LIN {X 0,Y 161.237,Z 153.823,A -85,B 0,C 180,E1 -25905.444,E2 -25905.444} C_VEL
LIN {X 0,Y 158.959,Z 150.146,A -85,B 0,C 180,E1 -25908.846,E2 -25908.846} C_VEL
LIN {X 0,Y 156.887,Z 147.156,A -85,B 0,C 180,E1 -25912.883,E2 -25912.883} C_VEL
LIN {X 0,Y 156.329,Z 145.593,A -85,B 0,C 180,E1 -25914.517,E2 -25914.517} C_VEL
LIN {X 0,Y 154.928,Z 144.258,A -85,B 0,C 180,E1 -25919.999,E2 -25919.999} C_VEL
LIN {X 0,Y 154.751,Z 144.476,A -85,B 0,C 180,E1 -25925.211,E2 -25925.211} C_VEL
LIN {X 0,Y 156.305,Z 145.838,A -85,B 0,C 180,E1 -25931.923,E2 -25931.923} C_VEL
LIN {X 0,Y 158.287,Z 149.53,A -85,B 0,C 180,E1 -25936.483,E2 -25936.483} C_VEL
LIN {X 0,Y 159.389,Z 150.896,A -85,B 0,C 180,E1 -25938.299,E2 -25938.299} C_VEL
LIN {X 0,Y 161.903,Z 155.182,A -85,B 0,C 180,E1 -25941.881,E2 -25941.881} C_VEL
LIN {X 0,Y 164.505,Z 160.547,A -85,B 0,C 180,E1 -25945.01,E2 -25945.01} C_VEL
LIN {X 0,Y 167.627,Z 167.381,A -85,B 0,C 180,E1 -25948.21,E2 -25948.21} C_VEL
LIN {X 0,Y 171.486,Z 176.831,A -85,B 0,C 180,E1 -25951.653,E2 -25951.653} C_VEL
LIN {X 0,Y 174.833,Z 186.302,A -85,B 0,C 180,E1 -25954.344,E2 -25954.344} C_VEL
LIN {X 0,Y 172.854,Z 207.577,A -85,B 0,C 180,E1 -25955.092,E2 -25955.092} C_VEL
LIN {X 0,Y 170.404,Z 220.728,A -85,B 0,C 180,E1 -25955.779,E2 -25955.779} C_VEL
LIN {X 0,Y 167.271,Z 232.382,A -85,B 0,C 180,E1 -25956.695,E2 -25956.695} C_VEL
LIN {X 0,Y 162.827,Z 244.666,A -85,B 0,C 180,E1 -25958.027,E2 -25958.027} C_VEL
LIN {X 0,Y 157.562,Z 256.097,A -85,B 0,C 180,E1 -25959.696,E2 -25959.696} C_VEL
LIN {X 0,Y 151.989,Z 266.408,A -85,B 0,C 180,E1 -25961.786,E2 -25961.786} C_VEL
LIN {X 0,Y 146.595,Z 274.853,A -85,B 0,C 180,E1 -25964.017,E2 -25964.017} C_VEL
LIN {X 0,Y 139.883,Z 284.024,A -85,B 0,C 180,E1 -25967.291,E2 -25967.291} C_VEL
LIN {X 0,Y 133.694,Z 291.425,A -85,B 0,C 180,E1 -25970.889,E2 -25970.889} C_VEL
LIN {X 0,Y 128.246,Z 297.387,A -85,B 0,C 180,E1 -25974.87,E2 -25974.87} C_VEL
LIN {X 0,Y 123.535,Z 302.12,A -85,B 0,C 180,E1 -25979.201,E2 -25979.201} C_VEL
LIN {X 0,Y 119.473,Z 305.757,A -85,B 0,C 180,E1 -25983.819,E2 -25983.819} C_VEL
LIN {X 0,Y 116.246,Z 308.403,A -85,B 0,C 180,E1 -25988.73,E2 -25988.73} C_VEL
LIN {X 0,Y 114.629,Z 309.67,A -85,B 0,C 180,E1 -25992.147,E2 -25992.147} C_VEL
LIN {X 0,Y 113.509,Z 310.529,A -85,B 0,C 180,E1 -25995.66,E2 -25995.66} C_VEL
LIN {X 0,Y 112.333,Z 311.033,A -85,B 0,C 180,E1 -26002.811,E2 -26002.811} C_VEL
LIN {X 0,Y 112.458,Z 310.179,A -85,B 0,C 180,E1 -26009.194,E2 -26009.194} C_VEL
LIN {X 0,Y 112.346,Z 308.795,A -85,B 0,C 180,E1 -26013.586,E2 -26013.586} C_VEL
LIN {X 0,Y 112.488,Z 306.212,A -85,B 0,C 180,E1 -26018.985,E2 -26018.985} C_VEL
LIN {X 0,Y 113.368,Z 302.594,A -85,B 0,C 180,E1 -26024.356,E2 -26024.356} C_VEL
LIN {X 0,Y 115.16,Z 297.853,A -85,B 0,C 180,E1 -26029.611,E2 -26029.611} C_VEL
LIN {X 0,Y 117.825,Z 291.844,A -85,B 0,C 180,E1 -26034.678,E2 -26034.678} C_VEL
LIN {X 0,Y 120.577,Z 286.067,A -85,B 0,C 180,E1 -26038.505,E2 -26038.505} C_VEL
LIN {X 0,Y 124.02,Z 278.346,A -85,B 0,C 180,E1 -26042.57,E2 -26042.57} C_VEL
LIN {X 0,Y 126.266,Z 273.338,A -85,B 0,C 180,E1 -26044.711,E2 -26044.711} C_VEL
LIN {X 0,Y 127.579,Z 269.067,A -85,B 0,C 180,E1 -26046.467,E2 -26046.467} C_VEL
LIN {X 0,Y 128.278,Z 261.803,A -85,B 0,C 180,E1 -26049.488,E2 -26049.488} C_VEL
LIN {X 0,Y 129.024,Z 254.081,A -85,B 0,C 180,E1 -26052.242,E2 -26052.242} C_VEL
LIN {X 0,Y 130.33,Z 249.097,A -85,B 0,C 180,E1 -26053.522,E2 -26053.522} C_VEL
LIN {X 0,Y 134.094,Z 237.597,A -85,B 0,C 180,E1 -26055.568,E2 -26055.568} C_VEL
LIN {X 0,Y 137.193,Z 225.349,A -85,B 0,C 180,E1 -26057.153,E2 -26057.153} C_VEL
LIN {X 0,Y 139.495,Z 212.87,A -85,B 0,C 180,E1 -26058.268,E2 -26058.268} C_VEL
LIN {X 0,Y 140.933,Z 199.169,A -85,B 0,C 180,E1 -26059.042,E2 -26059.042} C_VEL
LIN {X 0,Y 143.055,Z 169.052,A -85,B 0,C 180,E1 -26060.308,E2 -26060.308} C_VEL
LIN {X 0,Y 142.696,Z 161.497,A -85,B 0,C 180,E1 -26061.009,E2 -26061.009} C_VEL
LIN {X 0,Y 139.659,Z 152.428,A -85,B 0,C 180,E1 -26063.079,E2 -26063.079} C_VEL
LIN {X 0,Y 135.374,Z 142.008,A -85,B 0,C 180,E1 -26066.124,E2 -26066.124} C_VEL
LIN {X 0,Y 132.711,Z 136.591,A -85,B 0,C 180,E1 -26068.136,E2 -26068.136} C_VEL
LIN {X 0,Y 127.721,Z 129.053,A -85,B 0,C 180,E1 -26072.186,E2 -26072.186} C_VEL
LIN {X 0,Y 124.838,Z 124.988,A -85,B 0,C 180,E1 -26074.886,E2 -26074.886} C_VEL
LIN {X 0,Y 122.223,Z 121.297,A -85,B 0,C 180,E1 -26077.677,E2 -26077.677} C_VEL
LIN {X 0,Y 119.05,Z 117.651,A -85,B 0,C 180,E1 -26081.556,E2 -26081.556} C_VEL
LIN {X 0,Y 118.034,Z 115.687,A -85,B 0,C 180,E1 -26083.127,E2 -26083.127} C_VEL
LIN {X 0,Y 115.584,Z 113.816,A -85,B 0,C 180,E1 -26087.028,E2 -26087.028} C_VEL
LIN {X 0,Y 114.038,Z 110.593,A -85,B 0,C 180,E1 -26090.692,E2 -26090.692} C_VEL
LIN {X 0,Y 113.905,Z 110.069,A -85,B 0,C 180,E1 -26091.129,E2 -26091.129} C_VEL
LIN {X 0,Y 111.558,Z 108.57,A -85,B 0,C 180,E1 -26100.001,E2 -26100.001} C_VEL
LIN {X 0,Y 112.791,Z 109.816,A -85,B 0,C 180,E1 -26113.637,E2 -26113.637} C_VEL
LIN {X 0,Y 113.656,Z 110.24,A -85,B 0,C 180,E1 -26116.042,E2 -26116.042} C_VEL
LIN {X 0,Y 114.742,Z 112.902,A -85,B 0,C 180,E1 -26118.99,E2 -26118.99} C_VEL
LIN {X 0,Y 117.084,Z 115.281,A -85,B 0,C 180,E1 -26123.218,E2 -26123.218} C_VEL
LIN {X 0,Y 118.127,Z 115.966,A -85,B 0,C 180,E1 -26124.73,E2 -26124.73} C_VEL
LIN {X 0,Y 120.133,Z 119.302,A -85,B 0,C 180,E1 -26127.611,E2 -26127.611} C_VEL
LIN {X 0,Y 122.237,Z 121.386,A -85,B 0,C 180,E1 -26130.044,E2 -26130.044} C_VEL
LIN {X 0,Y 124.625,Z 124.868,A -85,B 0,C 180,E1 -26132.619,E2 -26132.619} C_VEL
LIN {X 0,Y 125.763,Z 126.328,A -85,B 0,C 180,E1 -26133.72,E2 -26133.72} C_VEL
LIN {X 0,Y 129.511,Z 131.842,A -85,B 0,C 180,E1 -26137.059,E2 -26137.059} C_VEL
LIN {X 0,Y 133.457,Z 137.926,A -85,B 0,C 180,E1 -26140.126,E2 -26140.126} C_VEL
LIN {X 0,Y 138.292,Z 146.234,A -85,B 0,C 180,E1 -26143.461,E2 -26143.461} C_VEL
LIN {X 0,Y 142.745,Z 155.217,A -85,B 0,C 180,E1 -26146.252,E2 -26146.252} C_VEL
LIN {X 0,Y 143.805,Z 157.638,A -85,B 0,C 180,E1 -26146.891,E2 -26146.891} C_VEL
LIN {X 0,Y 140.743,Z 198.449,A -85,B 0,C 180,E1 -26148.657,E2 -26148.657} C_VEL
LIN {X 0,Y 138.718,Z 212.325,A -85,B 0,C 180,E1 -26149.763,E2 -26149.763} C_VEL
LIN {X 0,Y 136.225,Z 224.495,A -85,B 0,C 180,E1 -26151.279,E2 -26151.279} C_VEL
LIN {X 0,Y 132.73,Z 237.021,A -85,B 0,C 180,E1 -26153.44,E2 -26153.44} C_VEL
LIN {X 0,Y 128.857,Z 248.183,A -85,B 0,C 180,E1 -26156.011,E2 -26156.011} C_VEL
LIN {X 0,Y 124.728,Z 258.248,A -85,B 0,C 180,E1 -26159.06,E2 -26159.06} C_VEL
LIN {X 0,Y 120.096,Z 268.136,A -85,B 0,C 180,E1 -26163.031,E2 -26163.031} C_VEL
LIN {X 0,Y 115.725,Z 276.841,A -85,B 0,C 180,E1 -26167.694,E2 -26167.694} C_VEL
LIN {X 0,Y 112.073,Z 283.795,A -85,B 0,C 180,E1 -26172.671,E2 -26172.671} C_VEL
LIN {X 0,Y 108.756,Z 290.167,A -85,B 0,C 180,E1 -26178.823,E2 -26178.823} C_VEL
LIN {X 0,Y 106.899,Z 294.363,A -85,B 0,C 180,E1 -26184.342,E2 -26184.342} C_VEL
LIN {X 0,Y 105.799,Z 297.516,A -85,B 0,C 180,E1 -26190.001,E2 -26190.001} C_VEL
LIN {X 0,Y 105.513,Z 299.091,A -85,B 0,C 180,E1 -26193.82,E2 -26193.82} C_VEL
LIN {X 0,Y 105.334,Z 300.263,A -85,B 0,C 180,E1 -26197.67,E2 -26197.67} C_VEL
LIN {X 0,Y 106.07,Z 301.363,A -85,B 0,C 180,E1 -26205.37,E2 -26205.37} C_VEL
LIN {X 0,Y 107.02,Z 301.338,A -85,B 0,C 180,E1 -26209.17,E2 -26209.17} C_VEL
LIN {X 0,Y 108.419,Z 300.902,A -85,B 0,C 180,E1 -26212.889,E2 -26212.889} C_VEL
LIN {X 0,Y 110.561,Z 299.844,A -85,B 0,C 180,E1 -26217.133,E2 -26217.133} C_VEL
LIN {X 0,Y 114.79,Z 297.11,A -85,B 0,C 180,E1 -26223.439,E2 -26223.439} C_VEL
LIN {X 0,Y 119.167,Z 293.727,A -85,B 0,C 180,E1 -26228.263,E2 -26228.263} C_VEL
LIN {X 0,Y 124.307,Z 289.239,A -85,B 0,C 180,E1 -26232.724,E2 -26232.724} C_VEL
LIN {X 0,Y 131.157,Z 282.378,A -85,B 0,C 180,E1 -26237.46,E2 -26237.46} C_VEL
LIN {X 0,Y 137.67,Z 274.904,A -85,B 0,C 180,E1 -26241.125,E2 -26241.125} C_VEL
LIN {X 0,Y 143.894,Z 266.42,A -85,B 0,C 180,E1 -26244.283,E2 -26244.283} C_VEL
LIN {X 0,Y 149.993,Z 256.814,A -85,B 0,C 180,E1 -26246.883,E2 -26246.883} C_VEL
LIN {X 0,Y 155.772,Z 246.135,A -85,B 0,C 180,E1 -26249.009,E2 -26249.009} C_VEL
LIN {X 0,Y 160.389,Z 235.789,A -85,B 0,C 180,E1 -26250.564,E2 -26250.564} C_VEL
LIN {X 0,Y 164.457,Z 224.001,A -85,B 0,C 180,E1 -26251.96,E2 -26251.96} C_VEL
LIN {X 0,Y 167.84,Z 211.19,A -85,B 0,C 180,E1 -26252.975,E2 -26252.975} C_VEL
LIN {X 0,Y 170.071,Z 198.637,A -85,B 0,C 180,E1 -26253.644,E2 -26253.644} C_VEL
LIN {X 0,Y 171.608,Z 182.647,A -85,B 0,C 180,E1 -26254.204,E2 -26254.204} C_VEL
LIN {X 0,Y 167.577,Z 174.242,A -85,B 0,C 180,E1 -26257.58,E2 -26257.58} C_VEL
LIN {X 0,Y 163.832,Z 167.391,A -85,B 0,C 180,E1 -26261.211,E2 -26261.211} C_VEL
LIN {X 0,Y 161.108,Z 162.795,A -85,B 0,C 180,E1 -26264.34,E2 -26264.34} C_VEL
LIN {X 0,Y 159.533,Z 160.138,A -85,B 0,C 180,E1 -26266.465,E2 -26266.465} C_VEL
LIN {X 0,Y 157.704,Z 156.967,A -85,B 0,C 180,E1 -26269.407,E2 -26269.407} C_VEL
LIN {X 0,Y 155.688,Z 153.841,A -85,B 0,C 180,E1 -26273.642,E2 -26273.642} C_VEL
LIN {X 0,Y 155.222,Z 152.527,A -85,B 0,C 180,E1 -26275.123,E2 -26275.123} C_VEL
LIN {X 0,Y 154.056,Z 151.337,A -85,B 0,C 180,E1 -26279.999,E2 -26279.999} C_VEL
LIN {X 0,Y 153.888,Z 151.51,A -85,B 0,C 180,E1 -26285.24,E2 -26285.24} C_VEL
LIN {X 0,Y 155.203,Z 152.67,A -85,B 0,C 180,E1 -26291.295,E2 -26291.295} C_VEL
LIN {X 0,Y 157.212,Z 156.507,A -85,B 0,C 180,E1 -26296.182,E2 -26296.182} C_VEL
LIN {X 0,Y 158.044,Z 157.648,A -85,B 0,C 180,E1 -26297.634,E2 -26297.634} C_VEL
LIN {X 0,Y 160.085,Z 161.28,A -85,B 0,C 180,E1 -26300.771,E2 -26300.771} C_VEL
LIN {X 0,Y 162.621,Z 166.938,A -85,B 0,C 180,E1 -26304.085,E2 -26304.085} C_VEL
LIN {X 0,Y 165.466,Z 173.642,A -85,B 0,C 180,E1 -26307.225,E2 -26307.225} C_VEL
LIN {X 0,Y 168.688,Z 182.087,A -85,B 0,C 180,E1 -26310.342,E2 -26310.342} C_VEL
LIN {X 0,Y 171.005,Z 188.932,A -85,B 0,C 180,E1 -26312.39,E2 -26312.39} C_VEL
LIN {X 0,Y 169.08,Z 208.154,A -85,B 0,C 180,E1 -26313.079,E2 -26313.079} C_VEL
LIN {X 0,Y 166.425,Z 221.664,A -85,B 0,C 180,E1 -26313.803,E2 -26313.803} C_VEL
LIN {X 0,Y 162.692,Z 234.387,A -85,B 0,C 180,E1 -26314.837,E2 -26314.837} C_VEL
LIN {X 0,Y 157.872,Z 246.668,A -85,B 0,C 180,E1 -26316.207,E2 -26316.207} C_VEL
LIN {X 0,Y 152.465,Z 257.651,A -85,B 0,C 180,E1 -26317.87,E2 -26317.87} C_VEL
LIN {X 0,Y 146.692,Z 267.553,A -85,B 0,C 180,E1 -26319.953,E2 -26319.953} C_VEL
LIN {X 0,Y 140.575,Z 276.564,A -85,B 0,C 180,E1 -26322.486,E2 -26322.486} C_VEL
LIN {X 0,Y 133.617,Z 285.378,A -85,B 0,C 180,E1 -26325.818,E2 -26325.818} C_VEL
LIN {X 0,Y 127.242,Z 292.459,A -85,B 0,C 180,E1 -26329.533,E2 -26329.533} C_VEL
LIN {X 0,Y 122.482,Z 297.278,A -85,B 0,C 180,E1 -26332.95,E2 -26332.95} C_VEL
LIN {X 0,Y 117.451,Z 301.965,A -85,B 0,C 180,E1 -26337.414,E2 -26337.414} C_VEL
LIN {X 0,Y 113.108,Z 305.56,A -85,B 0,C 180,E1 -26342.223,E2 -26342.223} C_VEL
LIN {X 0,Y 109.649,Z 308.167,A -85,B 0,C 180,E1 -26347.382,E2 -26347.382} C_VEL
LIN {X 0,Y 107.853,Z 309.412,A -85,B 0,C 180,E1 -26350.984,E2 -26350.984} C_VEL
LIN {X 0,Y 105.76,Z 310.659,A -85,B 0,C 180,E1 -26358.499,E2 -26358.499} C_VEL
LIN {X 0,Y 105.239,Z 310.367,A -85,B 0,C 180,E1 -26366.17,E2 -26366.17} C_VEL
LIN {X 0,Y 105.419,Z 309.613,A -85,B 0,C 180,E1 -26369.999,E2 -26369.999} C_VEL
LIN {X 0,Y 105.248,Z 308.39,A -85,B 0,C 180,E1 -26373.828,E2 -26373.828} C_VEL
LIN {X 0,Y 105.47,Z 305.767,A -85,B 0,C 180,E1 -26379.588,E2 -26379.588} C_VEL
LIN {X 0,Y 106.463,Z 302.106,A -85,B 0,C 180,E1 -26385.31,E2 -26385.31} C_VEL
LIN {X 0,Y 108.457,Z 297.32,A -85,B 0,C 180,E1 -26390.878,E2 -26390.878} C_VEL
LIN {X 0,Y 111.375,Z 291.262,A -85,B 0,C 180,E1 -26396.212,E2 -26396.212} C_VEL
LIN {X 0,Y 113.866,Z 286.445,A -85,B 0,C 180,E1 -26399.588,E2 -26399.588} C_VEL
LIN {X 0,Y 118.043,Z 277.64,A -85,B 0,C 180,E1 -26404.443,E2 -26404.443} C_VEL
LIN {X 0,Y 122.734,Z 267.649,A -85,B 0,C 180,E1 -26408.514,E2 -26408.514} C_VEL
LIN {X 0,Y 127.198,Z 257.535,A -85,B 0,C 180,E1 -26411.53,E2 -26411.53} C_VEL
LIN {X 0,Y 130.33,Z 249.097,A -85,B 0,C 180,E1 -26413.522,E2 -26413.522} C_VEL
LIN {X 0,Y 131.576,Z 243.979,A -85,B 0,C 180,E1 -26414.71,E2 -26414.71} C_VEL
LIN {X 0,Y 132.067,Z 235.477,A -85,B 0,C 180,E1 -26416.944,E2 -26416.944} C_VEL
LIN {X 0,Y 132.285,Z 226.668,A -85,B 0,C 180,E1 -26418.93,E2 -26418.93} C_VEL
LIN {X 0,Y 133.027,Z 221.072,A -85,B 0,C 180,E1 -26419.693,E2 -26419.693} C_VEL
LIN {X 0,Y 135.194,Z 207.663,A -85,B 0,C 180,E1 -26420.741,E2 -26420.741} C_VEL
LIN {X 0,Y 137.734,Z 177.242,A -85,B 0,C 180,E1 -26422.071,E2 -26422.071} C_VEL
LIN {X 0,Y 138.223,Z 169.25,A -85,B 0,C 180,E1 -26422.458,E2 -26422.458} C_VEL
LIN {X 0,Y 137.954,Z 163.915,A -85,B 0,C 180,E1 -26423.003,E2 -26423.003} C_VEL
LIN {X 0,Y 134.838,Z 154.473,A -85,B 0,C 180,E1 -26425.358,E2 -26425.358} C_VEL
LIN {X 0,Y 130.329,Z 143.432,A -85,B 0,C 180,E1 -26428.973,E2 -26428.973} C_VEL
LIN {X 0,Y 126.923,Z 137.867,A -85,B 0,C 180,E1 -26431.839,E2 -26431.839} C_VEL
LIN {X 0,Y 124.726,Z 134.478,A -85,B 0,C 180,E1 -26433.883,E2 -26433.883} C_VEL
LIN {X 0,Y 122.379,Z 130.942,A -85,B 0,C 180,E1 -26436.298,E2 -26436.298} C_VEL
LIN {X 0,Y 119.566,Z 127.012,A -85,B 0,C 180,E1 -26439.574,E2 -26439.574} C_VEL
LIN {X 0,Y 117.14,Z 123.924,A -85,B 0,C 180,E1 -26442.882,E2 -26442.882} C_VEL
LIN {X 0,Y 116.373,Z 122.439,A -85,B 0,C 180,E1 -26444.162,E2 -26444.162} C_VEL
LIN {X 0,Y 113.956,Z 120.189,A -85,B 0,C 180,E1 -26448.438,E2 -26448.438} C_VEL
LIN {X 0,Y 112.525,Z 116.989,A -85,B 0,C 180,E1 -26452.334,E2 -26452.334} C_VEL
LIN {X 0,Y 110.683,Z 115.663,A -85,B 0,C 180,E1 -26460.001,E2 -26460.001} C_VEL
LIN {X 0,Y 111.409,Z 116.622,A -85,B 0,C 180,E1 -26471.888,E2 -26471.888} C_VEL
LIN {X 0,Y 112.421,Z 117.245,A -85,B 0,C 180,E1 -26475.177,E2 -26475.177} C_VEL
LIN {X 0,Y 113.875,Z 120.333,A -85,B 0,C 180,E1 -26479.141,E2 -26479.141} C_VEL
LIN {X 0,Y 116.456,Z 122.726,A -85,B 0,C 180,E1 -26483.695,E2 -26483.695} C_VEL
LIN {X 0,Y 118.819,Z 126.398,A -85,B 0,C 180,E1 -26487.211,E2 -26487.211} C_VEL
LIN {X 0,Y 120.235,Z 127.963,A -85,B 0,C 180,E1 -26488.951,E2 -26488.951} C_VEL
LIN {X 0,Y 123.415,Z 132.552,A -85,B 0,C 180,E1 -26492.506,E2 -26492.506} C_VEL
LIN {X 0,Y 126.876,Z 137.847,A -85,B 0,C 180,E1 -26495.824,E2 -26495.824} C_VEL
LIN {X 0,Y 131.85,Z 145.96,A -85,B 0,C 180,E1 -26499.897,E2 -26499.897} C_VEL
LIN {X 0,Y 136.77,Z 155.402,A -85,B 0,C 180,E1 -26503.429,E2 -26503.429} C_VEL
LIN {X 0,Y 138.953,Z 160.638,A -85,B 0,C 180,E1 -26504.921,E2 -26504.921} C_VEL
LIN {X 0,Y 135.889,Z 198.312,A -85,B 0,C 180,E1 -26506.513,E2 -26506.513} C_VEL
LIN {X 0,Y 133.86,Z 211.948,A -85,B 0,C 180,E1 -26507.599,E2 -26507.599} C_VEL
LIN {X 0,Y 131.331,Z 223.788,A -85,B 0,C 180,E1 -26509.04,E2 -26509.04} C_VEL
LIN {X 0,Y 128.187,Z 235.014,A -85,B 0,C 180,E1 -26510.914,E2 -26510.914} C_VEL
LIN {X 0,Y 124.08,Z 246.604,A -85,B 0,C 180,E1 -26513.508,E2 -26513.508} C_VEL
LIN {X 0,Y 119.677,Z 257.032,A -85,B 0,C 180,E1 -26516.597,E2 -26516.597} C_VEL
LIN {X 0,Y 115.532,Z 265.569,A -85,B 0,C 180,E1 -26519.878,E2 -26519.878} C_VEL
LIN {X 0,Y 111.435,Z 273.431,A -85,B 0,C 180,E1 -26523.803,E2 -26523.803} C_VEL
LIN {X 0,Y 107.183,Z 281.123,A -85,B 0,C 180,E1 -26528.862,E2 -26528.862} C_VEL
LIN {X 0,Y 103.644,Z 287.295,A -85,B 0,C 180,E1 -26534.263,E2 -26534.263} C_VEL
LIN {X 0,Y 101.061,Z 292.199,A -85,B 0,C 180,E1 -26539.989,E2 -26539.989} C_VEL
LIN {X 0,Y 99.392,Z 295.99,A -85,B 0,C 180,E1 -26545.946,E2 -26545.946} C_VEL
LIN {X 0,Y 98.505,Z 299.016,A -85,B 0,C 180,E1 -26552.721,E2 -26552.721} C_VEL
LIN {X 0,Y 98.254,Z 300.638,A -85,B 0,C 180,E1 -26558.226,E2 -26558.226} C_VEL
LIN {X 0,Y 99.154,Z 301.698,A -85,B 0,C 180,E1 -26566.472,E2 -26566.472} C_VEL
LIN {X 0,Y 100.279,Z 301.651,A -85,B 0,C 180,E1 -26570.514,E2 -26570.514} C_VEL
LIN {X 0,Y 101.83,Z 301.174,A -85,B 0,C 180,E1 -26574.464,E2 -26574.464} C_VEL
LIN {X 0,Y 103.939,Z 300.23,A -85,B 0,C 180,E1 -26578.474,E2 -26578.474} C_VEL
LIN {X 0,Y 108.832,Z 297.311,A -85,B 0,C 180,E1 -26585.536,E2 -26585.536} C_VEL
LIN {X 0,Y 113.601,Z 293.884,A -85,B 0,C 180,E1 -26590.512,E2 -26590.512} C_VEL
LIN {X 0,Y 119.112,Z 289.341,A -85,B 0,C 180,E1 -26595.077,E2 -26595.077} C_VEL
LIN {X 0,Y 126.396,Z 282.408,A -85,B 0,C 180,E1 -26599.868,E2 -26599.868} C_VEL
LIN {X 0,Y 133.257,Z 274.87,A -85,B 0,C 180,E1 -26603.543,E2 -26603.543} C_VEL
LIN {X 0,Y 139.538,Z 266.674,A -85,B 0,C 180,E1 -26606.558,E2 -26606.558} C_VEL
LIN {X 0,Y 146.184,Z 256.571,A -85,B 0,C 180,E1 -26609.247,E2 -26609.247} C_VEL
LIN {X 0,Y 152.193,Z 245.775,A -85,B 0,C 180,E1 -26611.33,E2 -26611.33} C_VEL
LIN {X 0,Y 156.988,Z 235.258,A -85,B 0,C 180,E1 -26612.845,E2 -26612.845} C_VEL
LIN {X 0,Y 161.354,Z 222.655,A -85,B 0,C 180,E1 -26614.255,E2 -26614.255} C_VEL
LIN {X 0,Y 164.701,Z 209.907,A -85,B 0,C 180,E1 -26615.201,E2 -26615.201} C_VEL
LIN {X 0,Y 166.847,Z 197.391,A -85,B 0,C 180,E1 -26615.818,E2 -26615.818} C_VEL
LIN {X 0,Y 167.953,Z 185.982,A -85,B 0,C 180,E1 -26616.214,E2 -26616.214} C_VEL
LIN {X 0,Y 164.549,Z 178.774,A -85,B 0,C 180,E1 -26619.376,E2 -26619.376} C_VEL
LIN {X 0,Y 161.215,Z 172.413,A -85,B 0,C 180,E1 -26622.983,E2 -26622.983} C_VEL
LIN {X 0,Y 158.21,Z 166.998,A -85,B 0,C 180,E1 -26627.003,E2 -26627.003} C_VEL
LIN {X 0,Y 156.29,Z 163.6,A -85,B 0,C 180,E1 -26630.285,E2 -26630.285} C_VEL
LIN {X 0,Y 154.456,Z 160.326,A -85,B 0,C 180,E1 -26634.614,E2 -26634.614} C_VEL
LIN {X 0,Y 154.131,Z 159.461,A -85,B 0,C 180,E1 -26635.744,E2 -26635.744} C_VEL
LIN {X 0,Y 153.184,Z 158.412,A -85,B 0,C 180,E1 -26639.999,E2 -26639.999} C_VEL
LIN {X 0,Y 153.022,Z 158.562,A -85,B 0,C 180,E1 -26645.27,E2 -26645.27} C_VEL
LIN {X 0,Y 154.161,Z 159.663,A -85,B 0,C 180,E1 -26650.831,E2 -26650.831} C_VEL
LIN {X 0,Y 156.356,Z 163.745,A -85,B 0,C 180,E1 -26656.273,E2 -26656.273} C_VEL
LIN {X 0,Y 158.494,Z 167.806,A -85,B 0,C 180,E1 -26659.899,E2 -26659.899} C_VEL
LIN {X 0,Y 160.805,Z 173.342,A -85,B 0,C 180,E1 -26663.162,E2 -26663.162} C_VEL
LIN {X 0,Y 163.225,Z 179.624,A -85,B 0,C 180,E1 -26666.076,E2 -26666.076} C_VEL
LIN {X 0,Y 165.894,Z 187.063,A -85,B 0,C 180,E1 -26668.895,E2 -26668.895} C_VEL
LIN {X 0,Y 167.378,Z 191.61,A -85,B 0,C 180,E1 -26670.347,E2 -26670.347} C_VEL
LIN {X 0,Y 165.614,Z 208.192,A -85,B 0,C 180,E1 -26670.959,E2 -26670.959} C_VEL
LIN {X 0,Y 163.07,Z 220.692,A -85,B 0,C 180,E1 -26671.595,E2 -26671.595} C_VEL
LIN {X 0,Y 159.241,Z 233.657,A -85,B 0,C 180,E1 -26672.616,E2 -26672.616} C_VEL
LIN {X 0,Y 154.505,Z 245.511,A -85,B 0,C 180,E1 -26673.885,E2 -26673.885} C_VEL
LIN {X 0,Y 148.919,Z 256.669,A -85,B 0,C 180,E1 -26675.501,E2 -26675.501} C_VEL
LIN {X 0,Y 143.564,Z 265.704,A -85,B 0,C 180,E1 -26677.296,E2 -26677.296} C_VEL
LIN {X 0,Y 137.108,Z 274.997,A -85,B 0,C 180,E1 -26679.745,E2 -26679.745} C_VEL
LIN {X 0,Y 129.797,Z 284.018,A -85,B 0,C 180,E1 -26683.031,E2 -26683.031} C_VEL
LIN {X 0,Y 123.003,Z 291.307,A -85,B 0,C 180,E1 -26686.713,E2 -26686.713} C_VEL
LIN {X 0,Y 116.869,Z 297.169,A -85,B 0,C 180,E1 -26690.843,E2 -26690.843} C_VEL
LIN {X 0,Y 111.497,Z 301.81,A -85,B 0,C 180,E1 -26695.437,E2 -26695.437} C_VEL
LIN {X 0,Y 106.848,Z 305.363,A -85,B 0,C 180,E1 -26700.44,E2 -26700.44} C_VEL
LIN {X 0,Y 103.123,Z 307.931,A -85,B 0,C 180,E1 -26705.862,E2 -26705.862} C_VEL
LIN {X 0,Y 101.131,Z 309.149,A -85,B 0,C 180,E1 -26709.666,E2 -26709.666} C_VEL
LIN {X 0,Y 98.772,Z 310.346,A -85,B 0,C 180,E1 -26717.673,E2 -26717.673} C_VEL
LIN {X 0,Y 98.135,Z 310.016,A -85,B 0,C 180,E1 -26725.892,E2 -26725.892} C_VEL
LIN {X 0,Y 98.331,Z 309.227,A -85,B 0,C 180,E1 -26729.999,E2 -26729.999} C_VEL
LIN {X 0,Y 98.138,Z 307.982,A -85,B 0,C 180,E1 -26734.105,E2 -26734.105} C_VEL
LIN {X 0,Y 98.446,Z 305.32,A -85,B 0,C 180,E1 -26740.28,E2 -26740.28} C_VEL
LIN {X 0,Y 99.596,Z 301.615,A -85,B 0,C 180,E1 -26746.394,E2 -26746.394} C_VEL
LIN {X 0,Y 101.819,Z 296.784,A -85,B 0,C 180,E1 -26752.31,E2 -26752.31} C_VEL
LIN {X 0,Y 105.027,Z 290.676,A -85,B 0,C 180,E1 -26757.93,E2 -26757.93} C_VEL
LIN {X 0,Y 108.731,Z 283.676,A -85,B 0,C 180,E1 -26762.832,E2 -26762.832} C_VEL
LIN {X 0,Y 113.086,Z 275.286,A -85,B 0,C 180,E1 -26767.295,E2 -26767.295} C_VEL
LIN {X 0,Y 117.764,Z 265.812,A -85,B 0,C 180,E1 -26771.03,E2 -26771.03} C_VEL
LIN {X 0,Y 122.476,Z 255.299,A -85,B 0,C 180,E1 -26774.087,E2 -26774.087} C_VEL
LIN {X 0,Y 126.864,Z 243.589,A -85,B 0,C 180,E1 -26776.642,E2 -26776.642} C_VEL
LIN {X 0,Y 130.721,Z 231.132,A -85,B 0,C 180,E1 -26778.531,E2 -26778.531} C_VEL
LIN {X 0,Y 133.027,Z 221.072,A -85,B 0,C 180,E1 -26779.693,E2 -26779.693} C_VEL
LIN {X 0,Y 133.3,Z 217.293,A -85,B 0,C 180,E1 -26780.245,E2 -26780.245} C_VEL
LIN {X 0,Y 132.272,Z 211.412,A -85,B 0,C 180,E1 -26781.631,E2 -26781.631} C_VEL
LIN {X 0,Y 131.139,Z 205.471,A -85,B 0,C 180,E1 -26782.948,E2 -26782.948} C_VEL
LIN {X 0,Y 131.118,Z 201.6,A -85,B 0,C 180,E1 -26783.346,E2 -26783.346} C_VEL
LIN {X 0,Y 133.614,Z 170.677,A -85,B 0,C 180,E1 -26784.649,E2 -26784.649} C_VEL
LIN {X 0,Y 133.373,Z 166.236,A -85,B 0,C 180,E1 -26785.152,E2 -26785.152} C_VEL
LIN {X 0,Y 130.333,Z 156.897,A -85,B 0,C 180,E1 -26787.712,E2 -26787.712} C_VEL
LIN {X 0,Y 126.603,Z 147.597,A -85,B 0,C 180,E1 -26791.054,E2 -26791.054} C_VEL
LIN {X 0,Y 122.421,Z 140.695,A -85,B 0,C 180,E1 -26795.065,E2 -26795.065} C_VEL
LIN {X 0,Y 119.93,Z 136.833,A -85,B 0,C 180,E1 -26797.838,E2 -26797.838} C_VEL
LIN {X 0,Y 117.594,Z 133.386,A -85,B 0,C 180,E1 -26800.81,E2 -26800.81} C_VEL
LIN {X 0,Y 115.106,Z 129.816,A -85,B 0,C 180,E1 -26804.59,E2 -26804.59} C_VEL
LIN {X 0,Y 114.424,Z 128.9,A -85,B 0,C 180,E1 -26805.779,E2 -26805.779} C_VEL
LIN {X 0,Y 112.32,Z 126.391,A -85,B 0,C 180,E1 -26810.093,E2 -26810.093} C_VEL
LIN {X 0,Y 111.324,Z 123.921,A -85,B 0,C 180,E1 -26813.203,E2 -26813.203} C_VEL
LIN {X 0,Y 109.811,Z 122.733,A -85,B 0,C 180,E1 -26820.001,E2 -26820.001} C_VEL
LIN {X 0,Y 110.555,Z 123.691,A -85,B 0,C 180,E1 -26831.982,E2 -26831.982} C_VEL
LIN {X 0,Y 111.23,Z 124.124,A -85,B 0,C 180,E1 -26834.297,E2 -26834.297} C_VEL
LIN {X 0,Y 112.717,Z 127.319,A -85,B 0,C 180,E1 -26838.637,E2 -26838.637} C_VEL
LIN {X 0,Y 114.875,Z 129.481,A -85,B 0,C 180,E1 -26842.707,E2 -26842.707} C_VEL
LIN {X 0,Y 117.293,Z 133.205,A -85,B 0,C 180,E1 -26846.504,E2 -26846.504} C_VEL
LIN {X 0,Y 118.403,Z 134.67,A -85,B 0,C 180,E1 -26847.978,E2 -26847.978} C_VEL
LIN {X 0,Y 121.097,Z 138.712,A -85,B 0,C 180,E1 -26851.213,E2 -26851.213} C_VEL
LIN {X 0,Y 125.206,Z 145.238,A -85,B 0,C 180,E1 -26855.379,E2 -26855.379} C_VEL
LIN {X 0,Y 130.004,Z 153.951,A -85,B 0,C 180,E1 -26859.511,E2 -26859.511} C_VEL
LIN {X 0,Y 134.111,Z 162.58,A -85,B 0,C 180,E1 -26862.634,E2 -26862.634} C_VEL
LIN {X 0,Y 134.234,Z 163.049,A -85,B 0,C 180,E1 -26862.739,E2 -26862.739} C_VEL
LIN {X 0,Y 131.149,Z 198.863,A -85,B 0,C 180,E1 -26864.256,E2 -26864.256} C_VEL
LIN {X 0,Y 129.032,Z 212.339,A -85,B 0,C 180,E1 -26865.336,E2 -26865.336} C_VEL
LIN {X 0,Y 126.116,Z 225.223,A -85,B 0,C 180,E1 -26866.95,E2 -26866.95} C_VEL
LIN {X 0,Y 122.261,Z 237.726,A -85,B 0,C 180,E1 -26869.167,E2 -26869.167} C_VEL
LIN {X 0,Y 117.967,Z 248.875,A -85,B 0,C 180,E1 -26871.824,E2 -26871.824} C_VEL
LIN {X 0,Y 113.355,Z 258.928,A -85,B 0,C 180,E1 -26875.007,E2 -26875.007} C_VEL
LIN {X 0,Y 108.574,Z 268.002,A -85,B 0,C 180,E1 -26878.814,E2 -26878.814} C_VEL
LIN {X 0,Y 103.563,Z 276.836,A -85,B 0,C 180,E1 -26883.827,E2 -26883.827} C_VEL
LIN {X 0,Y 99.252,Z 283.95,A -85,B 0,C 180,E1 -26889.266,E2 -26889.266} C_VEL
LIN {X 0,Y 95.828,Z 289.621,A -85,B 0,C 180,E1 -26895.128,E2 -26895.128} C_VEL
LIN {X 0,Y 93.406,Z 294.088,A -85,B 0,C 180,E1 -26901.346,E2 -26901.346} C_VEL
LIN {X 0,Y 92.317,Z 296.449,A -85,B 0,C 180,E1 -26905.635,E2 -26905.635} C_VEL
LIN {X 0,Y 91.447,Z 299.258,A -85,B 0,C 180,E1 -26912.409,E2 -26912.409} C_VEL
LIN {X 0,Y 91.161,Z 301.015,A -85,B 0,C 180,E1 -26918.871,E2 -26918.871} C_VEL
LIN {X 0,Y 92.284,Z 302.033,A -85,B 0,C 180,E1 -26927.737,E2 -26927.737} C_VEL
LIN {X 0,Y 93.576,Z 301.958,A -85,B 0,C 180,E1 -26932.058,E2 -26932.058} C_VEL
LIN {X 0,Y 97.54,Z 300.537,A -85,B 0,C 180,E1 -26940.291,E2 -26940.291} C_VEL
LIN {X 0,Y 100.096,Z 299.235,A -85,B 0,C 180,E1 -26944.175,E2 -26944.175} C_VEL
LIN {X 0,Y 104.668,Z 296.447,A -85,B 0,C 180,E1 -26949.636,E2 -26949.636} C_VEL
LIN {X 0,Y 110.082,Z 292.612,A -85,B 0,C 180,E1 -26954.611,E2 -26954.611} C_VEL
LIN {X 0,Y 116.259,Z 287.62,A -85,B 0,C 180,E1 -26959.083,E2 -26959.083} C_VEL
LIN {X 0,Y 123.054,Z 281.31,A -85,B 0,C 180,E1 -26963.092,E2 -26963.092} C_VEL
LIN {X 0,Y 130.333,Z 273.36,A -85,B 0,C 180,E1 -26966.702,E2 -26966.702} C_VEL
LIN {X 0,Y 136.561,Z 265.338,A -85,B 0,C 180,E1 -26969.452,E2 -26969.452} C_VEL
LIN {X 0,Y 143.322,Z 255.26,A -85,B 0,C 180,E1 -26971.966,E2 -26971.966} C_VEL
LIN {X 0,Y 149.604,Z 243.987,A -85,B 0,C 180,E1 -26973.956,E2 -26973.956} C_VEL
LIN {X 0,Y 154.542,Z 232.884,A -85,B 0,C 180,E1 -26975.442,E2 -26975.442} C_VEL
LIN {X 0,Y 158.501,Z 221.395,A -85,B 0,C 180,E1 -26976.626,E2 -26976.626} C_VEL
LIN {X 0,Y 161.818,Z 208.577,A -85,B 0,C 180,E1 -26977.495,E2 -26977.495} C_VEL
LIN {X 0,Y 163.957,Z 195.109,A -85,B 0,C 180,E1 -26978.101,E2 -26978.101} C_VEL
LIN {X 0,Y 164.492,Z 189.481,A -85,B 0,C 180,E1 -26978.313,E2 -26978.313} C_VEL
LIN {X 0,Y 161.512,Z 182.854,A -85,B 0,C 180,E1 -26981.445,E2 -26981.445} C_VEL
LIN {X 0,Y 158.46,Z 176.844,A -85,B 0,C 180,E1 -26985.224,E2 -26985.224} C_VEL
LIN {X 0,Y 156.415,Z 173.06,A -85,B 0,C 180,E1 -26988.334,E2 -26988.334} C_VEL
LIN {X 0,Y 155.073,Z 170.411,A -85,B 0,C 180,E1 -26990.872,E2 -26990.872} C_VEL
LIN {X 0,Y 153.299,Z 166.94,A -85,B 0,C 180,E1 -26995.48,E2 -26995.48} C_VEL
LIN {X 0,Y 152.965,Z 166.3,A -85,B 0,C 180,E1 -26996.707,E2 -26996.707} C_VEL
LIN {X 0,Y 152.313,Z 165.475,A -85,B 0,C 180,E1 -26999.999,E2 -26999.999} C_VEL
LIN {X 0,Y 152.157,Z 165.616,A -85,B 0,C 180,E1 -27005.3,E2 -27005.3} C_VEL
LIN {X 0,Y 153.142,Z 166.681,A -85,B 0,C 180,E1 -27010.41,E2 -27010.41} C_VEL
LIN {X 0,Y 155.415,Z 171.177,A -85,B 0,C 180,E1 -27016.269,E2 -27016.269} C_VEL
LIN {X 0,Y 156.892,Z 174.235,A -85,B 0,C 180,E1 -27018.928,E2 -27018.928} C_VEL
LIN {X 0,Y 158.654,Z 178.809,A -85,B 0,C 180,E1 -27021.692,E2 -27021.692} C_VEL
LIN {X 0,Y 161.082,Z 185.57,A -85,B 0,C 180,E1 -27024.918,E2 -27024.918} C_VEL
LIN {X 0,Y 163.683,Z 193.574,A -85,B 0,C 180,E1 -27027.922,E2 -27027.922} C_VEL
LIN {X 0,Y 163.97,Z 194.549,A -85,B 0,C 180,E1 -27028.236,E2 -27028.236} C_VEL
LIN {X 0,Y 162.256,Z 209.092,A -85,B 0,C 180,E1 -27028.787,E2 -27028.787} C_VEL
LIN {X 0,Y 159.484,Z 221.768,A -85,B 0,C 180,E1 -27029.441,E2 -27029.441} C_VEL
LIN {X 0,Y 155.552,Z 234.28,A -85,B 0,C 180,E1 -27030.426,E2 -27030.426} C_VEL
LIN {X 0,Y 150.677,Z 245.942,A -85,B 0,C 180,E1 -27031.653,E2 -27031.653} C_VEL
LIN {X 0,Y 144.924,Z 256.942,A -85,B 0,C 180,E1 -27033.223,E2 -27033.223} C_VEL
LIN {X 0,Y 139.383,Z 265.875,A -85,B 0,C 180,E1 -27034.977,E2 -27034.977} C_VEL
LIN {X 0,Y 132.681,Z 275.061,A -85,B 0,C 180,E1 -27037.387,E2 -27037.387} C_VEL
LIN {X 0,Y 125.049,Z 284.016,A -85,B 0,C 180,E1 -27040.646,E2 -27040.646} C_VEL
LIN {X 0,Y 117.918,Z 291.248,A -85,B 0,C 180,E1 -27044.338,E2 -27044.338} C_VEL
LIN {X 0,Y 111.425,Z 297.053,A -85,B 0,C 180,E1 -27048.525,E2 -27048.525} C_VEL
LIN {X 0,Y 105.702,Z 301.648,A -85,B 0,C 180,E1 -27053.243,E2 -27053.243} C_VEL
LIN {X 0,Y 100.713,Z 305.165,A -85,B 0,C 180,E1 -27058.44,E2 -27058.44} C_VEL
LIN {X 0,Y 96.653,Z 307.694,A -85,B 0,C 180,E1 -27064.132,E2 -27064.132} C_VEL
LIN {X 0,Y 94.473,Z 308.878,A -85,B 0,C 180,E1 -27068.162,E2 -27068.162} C_VEL
LIN {X 0,Y 91.82,Z 310.033,A -85,B 0,C 180,E1 -27076.724,E2 -27076.724} C_VEL
LIN {X 0,Y 91.054,Z 309.66,A -85,B 0,C 180,E1 -27085.572,E2 -27085.572} C_VEL
LIN {X 0,Y 91.224,Z 308.84,A -85,B 0,C 180,E1 -27089.999,E2 -27089.999} C_VEL
LIN {X 0,Y 91.057,Z 307.576,A -85,B 0,C 180,E1 -27094.425,E2 -27094.425} C_VEL
LIN {X 0,Y 91.424,Z 304.871,A -85,B 0,C 180,E1 -27101.079,E2 -27101.079} C_VEL
LIN {X 0,Y 92.757,Z 301.123,A -85,B 0,C 180,E1 -27107.641,E2 -27107.641} C_VEL
LIN {X 0,Y 95.259,Z 296.248,A -85,B 0,C 180,E1 -27113.938,E2 -27113.938} C_VEL
LIN {X 0,Y 98.793,Z 290.092,A -85,B 0,C 180,E1 -27119.864,E2 -27119.864} C_VEL
LIN {X 0,Y 102.993,Z 282.694,A -85,B 0,C 180,E1 -27125.211,E2 -27125.211} C_VEL
LIN {X 0,Y 107.485,Z 274.566,A -85,B 0,C 180,E1 -27129.605,E2 -27129.605} C_VEL
LIN {X 0,Y 112.507,Z 264.989,A -85,B 0,C 180,E1 -27133.403,E2 -27133.403} C_VEL
LIN {X 0,Y 117.436,Z 254.363,A -85,B 0,C 180,E1 -27136.519,E2 -27136.519} C_VEL
LIN {X 0,Y 122.099,Z 242.483,A -85,B 0,C 180,E1 -27139.065,E2 -27139.065} C_VEL
LIN {X 0,Y 126.115,Z 229.742,A -85,B 0,C 180,E1 -27140.958,E2 -27140.958} C_VEL
LIN {X 0,Y 129.046,Z 216.547,A -85,B 0,C 180,E1 -27142.389,E2 -27142.389} C_VEL
LIN {X 0,Y 130.914,Z 203.623,A -85,B 0,C 180,E1 -27143.251,E2 -27143.251} C_VEL
LIN {X 0,Y 131.118,Z 201.6,A -85,B 0,C 180,E1 -27143.346,E2 -27143.346} C_VEL
LIN {X 0,Y 131.421,Z 195.791,A -85,B 0,C 180,E1 -27143.736,E2 -27143.736} C_VEL
LIN {X 0,Y 130.759,Z 186.336,A -85,B 0,C 180,E1 -27144.902,E2 -27144.902} C_VEL
LIN {X 0,Y 129.204,Z 171.254,A -85,B 0,C 180,E1 -27147.075,E2 -27147.075} C_VEL
LIN {X 0,Y 128.985,Z 168.615,A -85,B 0,C 180,E1 -27147.449,E2 -27147.449} C_VEL
LIN {X 0,Y 126.052,Z 159.434,A -85,B 0,C 180,E1 -27150.228,E2 -27150.228} C_VEL
LIN {X 0,Y 123.46,Z 152.711,A -85,B 0,C 180,E1 -27152.831,E2 -27152.831} C_VEL
LIN {X 0,Y 119.657,Z 146.12,A -85,B 0,C 180,E1 -27156.873,E2 -27156.873} C_VEL
LIN {X 0,Y 117.337,Z 142.403,A -85,B 0,C 180,E1 -27159.741,E2 -27159.741} C_VEL
LIN {X 0,Y 115.636,Z 139.684,A -85,B 0,C 180,E1 -27162.153,E2 -27162.153} C_VEL
LIN {X 0,Y 113.166,Z 135.791,A -85,B 0,C 180,E1 -27166.359,E2 -27166.359} C_VEL
LIN {X 0,Y 111.047,Z 133.168,A -85,B 0,C 180,E1 -27170.998,E2 -27170.998} C_VEL
LIN {X 0,Y 110.165,Z 130.833,A -85,B 0,C 180,E1 -27174.05,E2 -27174.05} C_VEL
LIN {X 0,Y 108.94,Z 129.797,A -85,B 0,C 180,E1 -27180.001,E2 -27180.001} C_VEL
LIN {X 0,Y 109.702,Z 130.759,A -85,B 0,C 180,E1 -27192.076,E2 -27192.076} C_VEL
LIN {X 0,Y 110.101,Z 131.191,A -85,B 0,C 180,E1 -27193.582,E2 -27193.582} C_VEL
LIN {X 0,Y 111.99,Z 134.808,A -85,B 0,C 180,E1 -27199.071,E2 -27199.071} C_VEL
LIN {X 0,Y 113.332,Z 136.208,A -85,B 0,C 180,E1 -27201.689,E2 -27201.689} C_VEL
LIN {X 0,Y 115.942,Z 140.145,A -85,B 0,C 180,E1 -27205.994,E2 -27205.994} C_VEL
LIN {X 0,Y 119.101,Z 145.305,A -85,B 0,C 180,E1 -27210.183,E2 -27210.183} C_VEL
LIN {X 0,Y 122.443,Z 150.921,A -85,B 0,C 180,E1 -27213.856,E2 -27213.856} C_VEL
LIN {X 0,Y 126.682,Z 159.028,A -85,B 0,C 180,E1 -27217.86,E2 -27217.86} C_VEL
LIN {X 0,Y 129.632,Z 165.459,A -85,B 0,C 180,E1 -27220.35,E2 -27220.35} C_VEL
LIN {X 0,Y 126.61,Z 199.518,A -85,B 0,C 180,E1 -27221.842,E2 -27221.842} C_VEL
LIN {X 0,Y 124.431,Z 212.715,A -85,B 0,C 180,E1 -27222.906,E2 -27222.906} C_VEL
LIN {X 0,Y 121.362,Z 225.581,A -85,B 0,C 180,E1 -27224.521,E2 -27224.521} C_VEL
LIN {X 0,Y 117.603,Z 237.289,A -85,B 0,C 180,E1 -27226.589,E2 -27226.589} C_VEL
LIN {X 0,Y 113.073,Z 248.576,A -85,B 0,C 180,E1 -27229.262,E2 -27229.262} C_VEL
LIN {X 0,Y 108.178,Z 258.77,A -85,B 0,C 180,E1 -27232.479,E2 -27232.479} C_VEL
LIN {X 0,Y 102.603,Z 268.743,A -85,B 0,C 180,E1 -27236.773,E2 -27236.773} C_VEL
LIN {X 0,Y 97.272,Z 277.507,A -85,B 0,C 180,E1 -27241.991,E2 -27241.991} C_VEL
LIN {X 0,Y 92.661,Z 284.54,A -85,B 0,C 180,E1 -27247.715,E2 -27247.715} C_VEL
LIN {X 0,Y 89.003,Z 290.15,A -85,B 0,C 180,E1 -27253.958,E2 -27253.958} C_VEL
LIN {X 0,Y 86.423,Z 294.568,A -85,B 0,C 180,E1 -27260.641,E2 -27260.641} C_VEL
LIN {X 0,Y 85.247,Z 296.908,A -85,B 0,C 180,E1 -27265.272,E2 -27265.272} C_VEL
LIN {X 0,Y 84.382,Z 299.441,A -85,B 0,C 180,E1 -27271.849,E2 -27271.849} C_VEL
LIN {X 0,Y 84.104,Z 301.39,A -85,B 0,C 180,E1 -27279.622,E2 -27279.622} C_VEL
LIN {X 0,Y 85.465,Z 302.369,A -85,B 0,C 180,E1 -27289.205,E2 -27289.205} C_VEL
LIN {X 0,Y 86.958,Z 302.257,A -85,B 0,C 180,E1 -27293.837,E2 -27293.837} C_VEL
LIN {X 0,Y 91.388,Z 300.788,A -85,B 0,C 180,E1 -27302.571,E2 -27302.571} C_VEL
LIN {X 0,Y 94.217,Z 299.465,A -85,B 0,C 180,E1 -27306.639,E2 -27306.639} C_VEL
LIN {X 0,Y 99.211,Z 296.633,A -85,B 0,C 180,E1 -27312.298,E2 -27312.298} C_VEL
LIN {X 0,Y 105.069,Z 292.752,A -85,B 0,C 180,E1 -27317.375,E2 -27317.375} C_VEL
LIN {X 0,Y 111.684,Z 287.709,A -85,B 0,C 180,E1 -27321.87,E2 -27321.87} C_VEL
LIN {X 0,Y 118.871,Z 281.319,A -85,B 0,C 180,E1 -27325.868,E2 -27325.868} C_VEL
LIN {X 0,Y 126.513,Z 273.297,A -85,B 0,C 180,E1 -27329.436,E2 -27329.436} C_VEL
LIN {X 0,Y 133.003,Z 265.261,A -85,B 0,C 180,E1 -27332.102,E2 -27332.102} C_VEL
LIN {X 0,Y 140.1,Z 255.019,A -85,B 0,C 180,E1 -27334.552,E2 -27334.552} C_VEL
LIN {X 0,Y 145.861,Z 245.005,A -85,B 0,C 180,E1 -27336.276,E2 -27336.276} C_VEL
LIN {X 0,Y 150.964,Z 234.07,A -85,B 0,C 180,E1 -27337.711,E2 -27337.711} C_VEL
LIN {X 0,Y 155.13,Z 222.575,A -85,B 0,C 180,E1 -27338.881,E2 -27338.881} C_VEL
LIN {X 0,Y 158.682,Z 209.526,A -85,B 0,C 180,E1 -27339.765,E2 -27339.765} C_VEL
LIN {X 0,Y 160.808,Z 197.238,A -85,B 0,C 180,E1 -27340.318,E2 -27340.318} C_VEL
LIN {X 0,Y 161.238,Z 192.932,A -85,B 0,C 180,E1 -27340.524,E2 -27340.524} C_VEL
LIN {X 0,Y 158.139,Z 186.009,A -85,B 0,C 180,E1 -27344.286,E2 -27344.286} C_VEL
LIN {X 0,Y 155.514,Z 180.535,A -85,B 0,C 180,E1 -27348.266,E2 -27348.266} C_VEL
LIN {X 0,Y 153.719,Z 177.045,A -85,B 0,C 180,E1 -27351.785,E2 -27351.785} C_VEL
LIN {X 0,Y 152.096,Z 173.368,A -85,B 0,C 180,E1 -27356.688,E2 -27356.688} C_VEL
LIN {X 0,Y 151.441,Z 172.557,A -85,B 0,C 180,E1 -27359.999,E2 -27359.999} C_VEL
LIN {X 0,Y 151.215,Z 172.541,A -85,B 0,C 180,E1 -27363.997,E2 -27363.997} C_VEL
LIN {X 0,Y 152.097,Z 173.547,A -85,B 0,C 180,E1 -27369.81,E2 -27369.81} C_VEL
LIN {X 0,Y 154.157,Z 178.001,A -85,B 0,C 180,E1 -27375.62,E2 -27375.62} C_VEL
LIN {X 0,Y 155.35,Z 180.626,A -85,B 0,C 180,E1 -27377.95,E2 -27377.95} C_VEL
LIN {X 0,Y 157.282,Z 186.151,A -85,B 0,C 180,E1 -27381.232,E2 -27381.232} C_VEL
LIN {X 0,Y 159.801,Z 194.096,A -85,B 0,C 180,E1 -27384.782,E2 -27384.782} C_VEL
LIN {X 0,Y 160.807,Z 197.61,A -85,B 0,C 180,E1 -27386.064,E2 -27386.064} C_VEL
LIN {X 0,Y 158.919,Z 211.123,A -85,B 0,C 180,E1 -27386.59,E2 -27386.59} C_VEL
LIN {X 0,Y 156.124,Z 222.754,A -85,B 0,C 180,E1 -27387.196,E2 -27387.196} C_VEL
LIN {X 0,Y 152.095,Z 234.906,A -85,B 0,C 180,E1 -27388.129,E2 -27388.129} C_VEL
LIN {X 0,Y 147.093,Z 246.375,A -85,B 0,C 180,E1 -27389.31,E2 -27389.31} C_VEL
LIN {X 0,Y 141.173,Z 257.187,A -85,B 0,C 180,E1 -27390.821,E2 -27390.821} C_VEL
LIN {X 0,Y 134.039,Z 267.977,A -85,B 0,C 180,E1 -27392.972,E2 -27392.972} C_VEL
LIN {X 0,Y 127.164,Z 276.757,A -85,B 0,C 180,E1 -27395.392,E2 -27395.392} C_VEL
LIN {X 0,Y 119.266,Z 285.329,A -85,B 0,C 180,E1 -27398.666,E2 -27398.666} C_VEL
LIN {X 0,Y 111.881,Z 292.21,A -85,B 0,C 180,E1 -27402.429,E2 -27402.429} C_VEL
LIN {X 0,Y 104.085,Z 298.557,A -85,B 0,C 180,E1 -27407.527,E2 -27407.527} C_VEL
LIN {X 0,Y 98.233,Z 302.737,A -85,B 0,C 180,E1 -27412.544,E2 -27412.544} C_VEL
LIN {X 0,Y 93.115,Z 305.875,A -85,B 0,C 180,E1 -27418.105,E2 -27418.105} C_VEL
LIN {X 0,Y 90.288,Z 307.457,A -85,B 0,C 180,E1 -27422.156,E2 -27422.156} C_VEL
LIN {X 0,Y 87.89,Z 308.603,A -85,B 0,C 180,E1 -27426.432,E2 -27426.432} C_VEL
LIN {X 0,Y 84.908,Z 309.721,A -85,B 0,C 180,E1 -27435.621,E2 -27435.621} C_VEL
LIN {X 0,Y 84.17,Z 309.71,A -85,B 0,C 180,E1 -27440.385,E2 -27440.385} C_VEL
LIN {X 0,Y 83.972,Z 309.297,A -85,B 0,C 180,E1 -27445.198,E2 -27445.198} C_VEL
LIN {X 0,Y 84.135,Z 308.453,A -85,B 0,C 180,E1 -27449.999,E2 -27449.999} C_VEL
LIN {X 0,Y 83.974,Z 307.17,A -85,B 0,C 180,E1 -27454.799,E2 -27454.799} C_VEL
LIN {X 0,Y 84.44,Z 304.423,A -85,B 0,C 180,E1 -27462.008,E2 -27462.008} C_VEL
LIN {X 0,Y 85.955,Z 300.631,A -85,B 0,C 180,E1 -27469.089,E2 -27469.089} C_VEL
LIN {X 0,Y 88.792,Z 295.713,A -85,B 0,C 180,E1 -27475.805,E2 -27475.805} C_VEL
LIN {X 0,Y 92.689,Z 289.507,A -85,B 0,C 180,E1 -27482.055,E2 -27482.055} C_VEL
LIN {X 0,Y 97.226,Z 282.047,A -85,B 0,C 180,E1 -27487.646,E2 -27487.646} C_VEL
LIN {X 0,Y 102.077,Z 273.828,A -85,B 0,C 180,E1 -27492.165,E2 -27492.165} C_VEL
LIN {X 0,Y 107.436,Z 264.161,A -85,B 0,C 180,E1 -27496.018,E2 -27496.018} C_VEL
LIN {X 0,Y 112.609,Z 253.422,A -85,B 0,C 180,E1 -27499.175,E2 -27499.175} C_VEL
LIN {X 0,Y 116.914,Z 243.044,A -85,B 0,C 180,E1 -27501.393,E2 -27501.393} C_VEL
LIN {X 0,Y 121.107,Z 230.625,A -85,B 0,C 180,E1 -27503.278,E2 -27503.278} C_VEL
LIN {X 0,Y 124.346,Z 217.041,A -85,B 0,C 180,E1 -27504.78,E2 -27504.78} C_VEL
LIN {X 0,Y 126.31,Z 204.704,A -85,B 0,C 180,E1 -27505.646,E2 -27505.646} C_VEL
LIN {X 0,Y 129.204,Z 171.254,A -85,B 0,C 180,E1 -27507.075,E2 -27507.075} C_VEL
LIN {X 0,Y 128.661,Z 167.726,A -85,B 0,C 180,E1 -27507.729,E2 -27507.729} C_VEL
LIN {X 0,Y 127.223,Z 164.006,A -85,B 0,C 180,E1 -27508.992,E2 -27508.992} C_VEL
LIN {X 0,Y 125.315,Z 161.011,A -85,B 0,C 180,E1 -27510.579,E2 -27510.579} C_VEL
LIN {X 0,Y 120.899,Z 156.336,A -85,B 0,C 180,E1 -27514.49,E2 -27514.49} C_VEL
LIN {X 0,Y 117.701,Z 152.697,A -85,B 0,C 180,E1 -27517.897,E2 -27517.897} C_VEL
LIN {X 0,Y 115.183,Z 148.413,A -85,B 0,C 180,E1 -27521.289,E2 -27521.289} C_VEL
LIN {X 0,Y 113.711,Z 145.932,A -85,B 0,C 180,E1 -27523.596,E2 -27523.596} C_VEL
LIN {X 0,Y 111.451,Z 142.288,A -85,B 0,C 180,E1 -27527.856,E2 -27527.856} C_VEL
LIN {X 0,Y 109.527,Z 139.263,A -85,B 0,C 180,E1 -27532.859,E2 -27532.859} C_VEL
LIN {X 0,Y 108.994,Z 137.77,A -85,B 0,C 180,E1 -27535.03,E2 -27535.03} C_VEL
LIN {X 0,Y 108.064,Z 136.894,A -85,B 0,C 180,E1 -27540.001,E2 -27540.001} C_VEL
LIN {X 0,Y 108.42,Z 137.545,A -85,B 0,C 180,E1 -27550.269,E2 -27550.269} C_VEL
LIN {X 0,Y 108.964,Z 138.062,A -85,B 0,C 180,E1 -27552.68,E2 -27552.68} C_VEL
LIN {X 0,Y 110.809,Z 141.717,A -85,B 0,C 180,E1 -27558.49,E2 -27558.49} C_VEL
LIN {X 0,Y 111.863,Z 142.972,A -85,B 0,C 180,E1 -27560.714,E2 -27560.714} C_VEL
LIN {X 0,Y 114.616,Z 147.543,A -85,B 0,C 180,E1 -27565.569,E2 -27565.569} C_VEL
LIN {X 0,Y 116.994,Z 151.616,A -85,B 0,C 180,E1 -27568.922,E2 -27568.922} C_VEL
LIN {X 0,Y 120.206,Z 157.458,A -85,B 0,C 180,E1 -27572.751,E2 -27572.751} C_VEL
LIN {X 0,Y 123.63,Z 164.413,A -85,B 0,C 180,E1 -27576.271,E2 -27576.271} C_VEL
LIN {X 0,Y 125.317,Z 168.263,A -85,B 0,C 180,E1 -27577.863,E2 -27577.863} C_VEL
LIN {X 0,Y 122.286,Z 200.343,A -85,B 0,C 180,E1 -27579.264,E2 -27579.264} C_VEL
LIN {X 0,Y 119.904,Z 213.837,A -85,B 0,C 180,E1 -27580.363,E2 -27580.363} C_VEL
LIN {X 0,Y 116.848,Z 225.928,A -85,B 0,C 180,E1 -27581.901,E2 -27581.901} C_VEL
LIN {X 0,Y 112.599,Z 238.415,A -85,B 0,C 180,E1 -27584.129,E2 -27584.129} C_VEL
LIN {X 0,Y 107.821,Z 249.557,A -85,B 0,C 180,E1 -27586.812,E2 -27586.812} C_VEL
LIN {X 0,Y 103.233,Z 258.58,A -85,B 0,C 180,E1 -27589.705,E2 -27589.705} C_VEL
LIN {X 0,Y 97.786,Z 267.861,A -85,B 0,C 180,E1 -27593.636,E2 -27593.636} C_VEL
LIN {X 0,Y 91.996,Z 276.825,A -85,B 0,C 180,E1 -27598.96,E2 -27598.96} C_VEL
LIN {X 0,Y 86.899,Z 284.063,A -85,B 0,C 180,E1 -27604.876,E2 -27604.876} C_VEL
LIN {X 0,Y 83.395,Z 288.958,A -85,B 0,C 180,E1 -27610.302,E2 -27610.302} C_VEL
LIN {X 0,Y 80.244,Z 293.71,A -85,B 0,C 180,E1 -27617.354,E2 -27617.354} C_VEL
LIN {X 0,Y 78.184,Z 297.365,A -85,B 0,C 180,E1 -27624.844,E2 -27624.844} C_VEL
LIN {X 0,Y 77.326,Z 299.619,A -85,B 0,C 180,E1 -27631.172,E2 -27631.172} C_VEL
LIN {X 0,Y 77.055,Z 301.765,A -85,B 0,C 180,E1 -27640.512,E2 -27640.512} C_VEL
LIN {X 0,Y 78.713,Z 302.703,A -85,B 0,C 180,E1 -27650.927,E2 -27650.927} C_VEL
LIN {X 0,Y 80.444,Z 302.55,A -85,B 0,C 180,E1 -27655.903,E2 -27655.903} C_VEL
LIN {X 0,Y 85.412,Z 301.04,A -85,B 0,C 180,E1 -27665.17,E2 -27665.17} C_VEL
LIN {X 0,Y 88.534,Z 299.693,A -85,B 0,C 180,E1 -27669.426,E2 -27669.426} C_VEL
LIN {X 0,Y 94.009,Z 296.82,A -85,B 0,C 180,E1 -27675.254,E2 -27675.254} C_VEL
LIN {X 0,Y 100.327,Z 292.891,A -85,B 0,C 180,E1 -27680.406,E2 -27680.406} C_VEL
LIN {X 0,Y 108.624,Z 286.787,A -85,B 0,C 180,E1 -27685.583,E2 -27685.583} C_VEL
LIN {X 0,Y 116.299,Z 280.088,A -85,B 0,C 180,E1 -27689.446,E2 -27689.446} C_VEL
LIN {X 0,Y 123.743,Z 272.411,A -85,B 0,C 180,E1 -27692.644,E2 -27692.644} C_VEL
LIN {X 0,Y 131.359,Z 263.08,A -85,B 0,C 180,E1 -27695.444,E2 -27695.444} C_VEL
LIN {X 0,Y 137.908,Z 253.561,A -85,B 0,C 180,E1 -27697.473,E2 -27697.473} C_VEL
LIN {X 0,Y 143.882,Z 243.148,A -85,B 0,C 180,E1 -27699.097,E2 -27699.097} C_VEL
LIN {X 0,Y 149.143,Z 231.689,A -85,B 0,C 180,E1 -27700.47,E2 -27700.47} C_VEL
LIN {X 0,Y 153.292,Z 219.797,A -85,B 0,C 180,E1 -27701.533,E2 -27701.533} C_VEL
LIN {X 0,Y 156.622,Z 206.634,A -85,B 0,C 180,E1 -27702.293,E2 -27702.293} C_VEL
LIN {X 0,Y 158.197,Z 196.805,A -85,B 0,C 180,E1 -27702.729,E2 -27702.729} C_VEL
LIN {X 0,Y 155.729,Z 190.853,A -85,B 0,C 180,E1 -27706.294,E2 -27706.294} C_VEL
LIN {X 0,Y 153.557,Z 186.091,A -85,B 0,C 180,E1 -27710.117,E2 -27710.117} C_VEL
LIN {X 0,Y 152.546,Z 183.866,A -85,B 0,C 180,E1 -27712.388,E2 -27712.388} C_VEL
LIN {X 0,Y 151.054,Z 180.282,A -85,B 0,C 180,E1 -27717.333,E2 -27717.333} C_VEL
LIN {X 0,Y 150.568,Z 179.637,A -85,B 0,C 180,E1 -27719.999,E2 -27719.999} C_VEL
LIN {X 0,Y 150.348,Z 179.593,A -85,B 0,C 180,E1 -27724.02,E2 -27724.02} C_VEL
LIN {X 0,Y 151.086,Z 180.464,A -85,B 0,C 180,E1 -27729.285,E2 -27729.285} C_VEL
LIN {X 0,Y 152.884,Z 184.709,A -85,B 0,C 180,E1 -27734.873,E2 -27734.873} C_VEL
LIN {X 0,Y 153.862,Z 187.11,A -85,B 0,C 180,E1 -27736.984,E2 -27736.984} C_VEL
LIN {X 0,Y 155.492,Z 192.306,A -85,B 0,C 180,E1 -27740.073,E2 -27740.073} C_VEL
LIN {X 0,Y 157.472,Z 199.298,A -85,B 0,C 180,E1 -27743.247,E2 -27743.247} C_VEL
LIN {X 0,Y 157.821,Z 200.712,A -85,B 0,C 180,E1 -27743.801,E2 -27743.801} C_VEL
LIN {X 0,Y 155.565,Z 214.069,A -85,B 0,C 180,E1 -27744.334,E2 -27744.334} C_VEL
LIN {X 0,Y 152.524,Z 225.375,A -85,B 0,C 180,E1 -27744.952,E2 -27744.952} C_VEL
LIN {X 0,Y 148.366,Z 236.837,A -85,B 0,C 180,E1 -27745.837,E2 -27745.837} C_VEL
LIN {X 0,Y 143.002,Z 248.213,A -85,B 0,C 180,E1 -27747.028,E2 -27747.028} C_VEL
LIN {X 0,Y 136.169,Z 259.774,A -85,B 0,C 180,E1 -27748.666,E2 -27748.666} C_VEL
LIN {X 0,Y 128.861,Z 270.013,A -85,B 0,C 180,E1 -27750.794,E2 -27750.794} C_VEL
LIN {X 0,Y 121.802,Z 278.357,A -85,B 0,C 180,E1 -27753.21,E2 -27753.21} C_VEL
LIN {X 0,Y 113.62,Z 286.537,A -85,B 0,C 180,E1 -27756.473,E2 -27756.473} C_VEL
LIN {X 0,Y 105.966,Z 293.142,A -85,B 0,C 180,E1 -27760.294,E2 -27760.294} C_VEL
LIN {X 0,Y 98.944,Z 298.428,A -85,B 0,C 180,E1 -27764.739,E2 -27764.739} C_VEL
LIN {X 0,Y 92.661,Z 302.563,A -85,B 0,C 180,E1 -27769.855,E2 -27769.855} C_VEL
LIN {X 0,Y 87.142,Z 305.659,A -85,B 0,C 180,E1 -27775.627,E2 -27775.627} C_VEL
LIN {X 0,Y 84.051,Z 307.216,A -85,B 0,C 180,E1 -27779.886,E2 -27779.886} C_VEL
LIN {X 0,Y 81.402,Z 308.328,A -85,B 0,C 180,E1 -27784.424,E2 -27784.424} C_VEL
LIN {X 0,Y 78.012,Z 309.408,A -85,B 0,C 180,E1 -27794.318,E2 -27794.318} C_VEL
LIN {X 0,Y 77.171,Z 309.378,A -85,B 0,C 180,E1 -27799.504,E2 -27799.504} C_VEL
LIN {X 0,Y 76.886,Z 308.928,A -85,B 0,C 180,E1 -27804.754,E2 -27804.754} C_VEL
LIN {X 0,Y 77.05,Z 308.068,A -85,B 0,C 180,E1 -27809.998,E2 -27809.998} C_VEL
LIN {X 0,Y 76.888,Z 306.763,A -85,B 0,C 180,E1 -27815.243,E2 -27815.243} C_VEL
LIN {X 0,Y 77.46,Z 303.974,A -85,B 0,C 180,E1 -27823.109,E2 -27823.109} C_VEL
LIN {X 0,Y 79.222,Z 300.138,A -85,B 0,C 180,E1 -27830.783,E2 -27830.783} C_VEL
LIN {X 0,Y 82.41,Z 295.174,A -85,B 0,C 180,E1 -27837.971,E2 -27837.971} C_VEL
LIN {X 0,Y 86.735,Z 288.921,A -85,B 0,C 180,E1 -27844.554,E2 -27844.554} C_VEL
LIN {X 0,Y 90.919,Z 282.5,A -85,B 0,C 180,E1 -27849.621,E2 -27849.621} C_VEL
LIN {X 0,Y 95.837,Z 274.803,A -85,B 0,C 180,E1 -27854.158,E2 -27854.158} C_VEL
LIN {X 0,Y 101.418,Z 265.479,A -85,B 0,C 180,E1 -27858.153,E2 -27858.153} C_VEL
LIN {X 0,Y 106.865,Z 255.091,A -85,B 0,C 180,E1 -27861.347,E2 -27861.347} C_VEL
LIN {X 0,Y 111.955,Z 243.557,A -85,B 0,C 180,E1 -27863.922,E2 -27863.922} C_VEL
LIN {X 0,Y 116.31,Z 231.49,A -85,B 0,C 180,E1 -27865.797,E2 -27865.797} C_VEL
LIN {X 0,Y 119.738,Z 218.154,A -85,B 0,C 180,E1 -27867.294,E2 -27867.294} C_VEL
LIN {X 0,Y 122.022,Z 204.954,A -85,B 0,C 180,E1 -27868.248,E2 -27868.248} C_VEL
LIN {X 0,Y 125.03,Z 172.457,A -85,B 0,C 180,E1 -27869.61,E2 -27869.61} C_VEL
LIN {X 0,Y 123.767,Z 167.485,A -85,B 0,C 180,E1 -27871.003,E2 -27871.003} C_VEL
LIN {X 0,Y 120.684,Z 158.238,A -85,B 0,C 180,E1 -27874.443,E2 -27874.443} C_VEL
LIN {X 0,Y 117.701,Z 152.697,A -85,B 0,C 180,E1 -27877.897,E2 -27877.897} C_VEL
LIN {X 0,Y 115.637,Z 150.578,A -85,B 0,C 180,E1 -27880.417,E2 -27880.417} C_VEL
LIN {X 0,Y 112.275,Z 149.074,A -85,B 0,C 180,E1 -27885.068,E2 -27885.068} C_VEL
LIN {X 0,Y 109.19,Z 147.631,A -85,B 0,C 180,E1 -27891.07,E2 -27891.07} C_VEL
LIN {X 0,Y 108.536,Z 146.547,A -85,B 0,C 180,E1 -27893.073,E2 -27893.073} C_VEL
LIN {X 0,Y 107.959,Z 144.738,A -85,B 0,C 180,E1 -27895.626,E2 -27895.626} C_VEL
LIN {X 0,Y 107.19,Z 143.979,A -85,B 0,C 180,E1 -27900.001,E2 -27900.001} C_VEL
LIN {X 0,Y 107.39,Z 144.516,A -85,B 0,C 180,E1 -27909.417,E2 -27909.417} C_VEL
LIN {X 0,Y 107.884,Z 145.016,A -85,B 0,C 180,E1 -27911.914,E2 -27911.914} C_VEL
LIN {X 0,Y 109.605,Z 148.592,A -85,B 0,C 180,E1 -27917.815,E2 -27917.815} C_VEL
LIN {X 0,Y 110.423,Z 149.75,A -85,B 0,C 180,E1 -27919.709,E2 -27919.709} C_VEL
LIN {X 0,Y 112.826,Z 154.003,A -85,B 0,C 180,E1 -27924.343,E2 -27924.343} C_VEL
LIN {X 0,Y 115.12,Z 158.206,A -85,B 0,C 180,E1 -27927.856,E2 -27927.856} C_VEL
LIN {X 0,Y 118.376,Z 164.691,A -85,B 0,C 180,E1 -27932.024,E2 -27932.024} C_VEL
LIN {X 0,Y 121.224,Z 171.184,A -85,B 0,C 180,E1 -27935.193,E2 -27935.193} C_VEL
LIN {X 0,Y 118.339,Z 200.449,A -85,B 0,C 180,E1 -27936.464,E2 -27936.464} C_VEL
LIN {X 0,Y 115.837,Z 214.001,A -85,B 0,C 180,E1 -27937.532,E2 -27937.532} C_VEL
LIN {X 0,Y 112.59,Z 226.278,A -85,B 0,C 180,E1 -27939.073,E2 -27939.073} C_VEL
LIN {X 0,Y 108.454,Z 237.97,A -85,B 0,C 180,E1 -27941.123,E2 -27941.123} C_VEL
LIN {X 0,Y 103.414,Z 249.252,A -85,B 0,C 180,E1 -27943.775,E2 -27943.775} C_VEL
LIN {X 0,Y 97.956,Z 259.437,A -85,B 0,C 180,E1 -27947.033,E2 -27947.033} C_VEL
LIN {X 0,Y 92.196,Z 268.596,A -85,B 0,C 180,E1 -27951.033,E2 -27951.033} C_VEL
LIN {X 0,Y 86.003,Z 277.493,A -85,B 0,C 180,E1 -27956.525,E2 -27956.525} C_VEL
LIN {X 0,Y 80.541,Z 284.67,A -85,B 0,C 180,E1 -27962.736,E2 -27962.736} C_VEL
LIN {X 0,Y 76.769,Z 289.51,A -85,B 0,C 180,E1 -27968.521,E2 -27968.521} C_VEL
LIN {X 0,Y 73.362,Z 294.212,A -85,B 0,C 180,E1 -27976.145,E2 -27976.145} C_VEL
LIN {X 0,Y 71.108,Z 297.823,A -85,B 0,C 180,E1 -27984.33,E2 -27984.33} C_VEL
LIN {X 0,Y 70.286,Z 299.868,A -85,B 0,C 180,E1 -27990.645,E2 -27990.645} C_VEL
LIN {X 0,Y 70.017,Z 302.141,A -85,B 0,C 180,E1 -28001.583,E2 -28001.583} C_VEL
LIN {X 0,Y 72.047,Z 303.032,A -85,B 0,C 180,E1 -28012.968,E2 -28012.968} C_VEL
LIN {X 0,Y 74.06,Z 302.842,A -85,B 0,C 180,E1 -28018.327,E2 -28018.327} C_VEL
LIN {X 0,Y 79.637,Z 301.291,A -85,B 0,C 180,E1 -28028.154,E2 -28028.154} C_VEL
LIN {X 0,Y 83.078,Z 299.913,A -85,B 0,C 180,E1 -28032.593,E2 -28032.593} C_VEL
LIN {X 0,Y 89.092,Z 296.999,A -85,B 0,C 180,E1 -28038.541,E2 -28038.541} C_VEL
LIN {X 0,Y 97.602,Z 291.897,A -85,B 0,C 180,E1 -28044.825,E2 -28044.825} C_VEL
LIN {X 0,Y 106.035,Z 285.841,A -85,B 0,C 180,E1 -28049.504,E2 -28049.504} C_VEL
LIN {X 0,Y 114.207,Z 278.832,A -85,B 0,C 180,E1 -28053.165,E2 -28053.165} C_VEL
LIN {X 0,Y 122.667,Z 270.007,A -85,B 0,C 180,E1 -28056.45,E2 -28056.45} C_VEL
LIN {X 0,Y 130.037,Z 260.934,A -85,B 0,C 180,E1 -28058.799,E2 -28058.799} C_VEL
LIN {X 0,Y 136.859,Z 250.891,A -85,B 0,C 180,E1 -28060.668,E2 -28060.668} C_VEL
LIN {X 0,Y 143.032,Z 239.668,A -85,B 0,C 180,E1 -28062.18,E2 -28062.18} C_VEL
LIN {X 0,Y 148.259,Z 227.435,A -85,B 0,C 180,E1 -28063.475,E2 -28063.475} C_VEL
LIN {X 0,Y 152.352,Z 214.688,A -85,B 0,C 180,E1 -28064.363,E2 -28064.363} C_VEL
LIN {X 0,Y 155.166,Z 201.655,A -85,B 0,C 180,E1 -28064.976,E2 -28064.976} C_VEL
LIN {X 0,Y 155.307,Z 200.68,A -85,B 0,C 180,E1 -28065.039,E2 -28065.039} C_VEL
LIN {X 0,Y 153.353,Z 195.438,A -85,B 0,C 180,E1 -28068.601,E2 -28068.601} C_VEL
LIN {X 0,Y 151.643,Z 191.265,A -85,B 0,C 180,E1 -28072.342,E2 -28072.342} C_VEL
LIN {X 0,Y 150.067,Z 187.236,A -85,B 0,C 180,E1 -28077.819,E2 -28077.819} C_VEL
LIN {X 0,Y 149.487,Z 186.51,A -85,B 0,C 180,E1 -28082.694,E2 -28082.694} C_VEL
LIN {X 0,Y 150.115,Z 187.51,A -85,B 0,C 180,E1 -28088.921,E2 -28088.921} C_VEL
LIN {X 0,Y 151.695,Z 191.554,A -85,B 0,C 180,E1 -28094.256,E2 -28094.256} C_VEL
LIN {X 0,Y 152.478,Z 193.804,A -85,B 0,C 180,E1 -28096.14,E2 -28096.14} C_VEL
LIN {X 0,Y 153.736,Z 198.332,A -85,B 0,C 180,E1 -28098.835,E2 -28098.835} C_VEL
LIN {X 0,Y 155.017,Z 203.925,A -85,B 0,C 180,E1 -28101.439,E2 -28101.439} C_VEL
LIN {X 0,Y 152.43,Z 216.706,A -85,B 0,C 180,E1 -28101.965,E2 -28101.965} C_VEL
LIN {X 0,Y 148.602,Z 229.309,A -85,B 0,C 180,E1 -28102.71,E2 -28102.71} C_VEL
LIN {X 0,Y 143.864,Z 240.883,A -85,B 0,C 180,E1 -28103.654,E2 -28103.654} C_VEL
LIN {X 0,Y 137.602,Z 252.683,A -85,B 0,C 180,E1 -28104.961,E2 -28104.961} C_VEL
LIN {X 0,Y 130.629,Z 263.255,A -85,B 0,C 180,E1 -28106.561,E2 -28106.561} C_VEL
LIN {X 0,Y 123.92,Z 271.899,A -85,B 0,C 180,E1 -28108.468,E2 -28108.468} C_VEL
LIN {X 0,Y 116.628,Z 279.879,A -85,B 0,C 180,E1 -28110.826,E2 -28110.826} C_VEL
LIN {X 0,Y 108.182,Z 287.722,A -85,B 0,C 180,E1 -28114.074,E2 -28114.074} C_VEL
LIN {X 0,Y 98.945,Z 294.921,A -85,B 0,C 180,E1 -28118.616,E2 -28118.616} C_VEL
LIN {X 0,Y 91.746,Z 299.762,A -85,B 0,C 180,E1 -28123.305,E2 -28123.305} C_VEL
LIN {X 0,Y 85.268,Z 303.5,A -85,B 0,C 180,E1 -28128.746,E2 -28128.746} C_VEL
LIN {X 0,Y 81.359,Z 305.444,A -85,B 0,C 180,E1 -28132.792,E2 -28132.792} C_VEL
LIN {X 0,Y 77.97,Z 306.968,A -85,B 0,C 180,E1 -28137.258,E2 -28137.258} C_VEL
LIN {X 0,Y 72.79,Z 308.763,A -85,B 0,C 180,E1 -28147.28,E2 -28147.28} C_VEL
LIN {X 0,Y 70.176,Z 309.041,A -85,B 0,C 180,E1 -28158.444,E2 -28158.444} C_VEL
LIN {X 0,Y 69.81,Z 308.559,A -85,B 0,C 180,E1 -28164.22,E2 -28164.22} C_VEL
LIN {X 0,Y 69.954,Z 307.68,A -85,B 0,C 180,E1 -28169.998,E2 -28169.998} C_VEL
LIN {X 0,Y 69.798,Z 306.355,A -85,B 0,C 180,E1 -28175.777,E2 -28175.777} C_VEL
LIN {X 0,Y 70.531,Z 303.524,A -85,B 0,C 180,E1 -28184.423,E2 -28184.423} C_VEL
LIN {X 0,Y 72.577,Z 299.643,A -85,B 0,C 180,E1 -28192.787,E2 -28192.787} C_VEL
LIN {X 0,Y 76.165,Z 294.634,A -85,B 0,C 180,E1 -28200.496,E2 -28200.496} C_VEL
LIN {X 0,Y 80.934,Z 288.328,A -85,B 0,C 180,E1 -28207.432,E2 -28207.432} C_VEL
LIN {X 0,Y 85.513,Z 281.849,A -85,B 0,C 180,E1 -28212.689,E2 -28212.689} C_VEL
LIN {X 0,Y 90.842,Z 274.088,A -85,B 0,C 180,E1 -28217.302,E2 -28217.302} C_VEL
LIN {X 0,Y 96.816,Z 264.647,A -85,B 0,C 180,E1 -28221.291,E2 -28221.291} C_VEL
LIN {X 0,Y 102.526,Z 254.14,A -85,B 0,C 180,E1 -28224.488,E2 -28224.488} C_VEL
LIN {X 0,Y 107.927,Z 242.479,A -85,B 0,C 180,E1 -28226.969,E2 -28226.969} C_VEL
LIN {X 0,Y 112.448,Z 230.078,A -85,B 0,C 180,E1 -28228.809,E2 -28228.809} C_VEL
LIN {X 0,Y 115.921,Z 216.716,A -85,B 0,C 180,E1 -28230.256,E2 -28230.256} C_VEL
LIN {X 0,Y 118.146,Z 204.07,A -85,B 0,C 180,E1 -28231.1,E2 -28231.1} C_VEL
LIN {X 0,Y 121.024,Z 174.257,A -85,B 0,C 180,E1 -28232.318,E2 -28232.318} C_VEL
LIN {X 0,Y 118.547,Z 165.626,A -85,B 0,C 180,E1 -28235.402,E2 -28235.402} C_VEL
LIN {X 0,Y 117.328,Z 162.434,A -85,B 0,C 180,E1 -28236.948,E2 -28236.948} C_VEL
LIN {X 0,Y 113.97,Z 155.835,A -85,B 0,C 180,E1 -28241.563,E2 -28241.563} C_VEL
LIN {X 0,Y 111.838,Z 152.185,A -85,B 0,C 180,E1 -28245.116,E2 -28245.116} C_VEL
LIN {X 0,Y 110.016,Z 148.953,A -85,B 0,C 180,E1 -28248.952,E2 -28248.952} C_VEL
LIN {X 0,Y 108.536,Z 146.547,A -85,B 0,C 180,E1 -28253.073,E2 -28253.073} C_VEL
LIN {X 0,Y 107.988,Z 145.755,A -85,B 0,C 180,E1 -28255.069,E2 -28255.069} C_VEL
LIN {X 0,Y 107.458,Z 145.804,A -85,B 0,C 180,E1 -28257.131,E2 -28257.131} C_VEL
LIN {X 0,Y 106.625,Z 147.498,A -85,B 0,C 180,E1 -28261.271,E2 -28261.271} C_VEL
LIN {X 0,Y 106.316,Z 151.052,A -85,B 0,C 180,E1 -28267.665,E2 -28267.665} C_VEL
LIN {X 0,Y 106.592,Z 151.621,A -85,B 0,C 180,E1 -28269.852,E2 -28269.852} C_VEL
LIN {X 0,Y 106.866,Z 152.11,A -85,B 0,C 180,E1 -28271.38,E2 -28271.38} C_VEL
LIN {X 0,Y 108.553,Z 155.61,A -85,B 0,C 180,E1 -28277.465,E2 -28277.465} C_VEL
LIN {X 0,Y 110.965,Z 160.191,A -85,B 0,C 180,E1 -28282.837,E2 -28282.837} C_VEL
LIN {X 0,Y 113.517,Z 165.282,A -85,B 0,C 180,E1 -28287.109,E2 -28287.109} C_VEL
LIN {X 0,Y 116.685,Z 172.395,A -85,B 0,C 180,E1 -28291.451,E2 -28291.451} C_VEL
LIN {X 0,Y 117.418,Z 174.416,A -85,B 0,C 180,E1 -28292.387,E2 -28292.387} C_VEL
LIN {X 0,Y 114.602,Z 201.085,A -85,B 0,C 180,E1 -28293.501,E2 -28293.501} C_VEL
LIN {X 0,Y 112.204,Z 213.626,A -85,B 0,C 180,E1 -28294.459,E2 -28294.459} C_VEL
LIN {X 0,Y 108.64,Z 226.624,A -85,B 0,C 180,E1 -28296.039,E2 -28296.039} C_VEL
LIN {X 0,Y 103.966,Z 239.095,A -85,B 0,C 180,E1 -28298.203,E2 -28298.203} C_VEL
LIN {X 0,Y 98.646,Z 250.236,A -85,B 0,C 180,E1 -28300.804,E2 -28300.804} C_VEL
LIN {X 0,Y 92.899,Z 260.268,A -85,B 0,C 180,E1 -28304.055,E2 -28304.055} C_VEL
LIN {X 0,Y 86.822,Z 269.332,A -85,B 0,C 180,E1 -28308.103,E2 -28308.103} C_VEL
LIN {X 0,Y 80.188,Z 278.161,A -85,B 0,C 180,E1 -28313.731,E2 -28313.731} C_VEL
LIN {X 0,Y 74.317,Z 285.267,A -85,B 0,C 180,E1 -28320.234,E2 -28320.234} C_VEL
LIN {X 0,Y 68.851,Z 291.729,A -85,B 0,C 180,E1 -28329.069,E2 -28329.069} C_VEL
LIN {X 0,Y 65.567,Z 296.005,A -85,B 0,C 180,E1 -28337.623,E2 -28337.623} C_VEL
LIN {X 0,Y 63.256,Z 300.006,A -85,B 0,C 180,E1 -28349.559,E2 -28349.559} C_VEL
LIN {X 0,Y 62.809,Z 301.511,A -85,B 0,C 180,E1 -28356.426,E2 -28356.426} C_VEL
LIN {X 0,Y 63.025,Z 302.516,A -85,B 0,C 180,E1 -28362.889,E2 -28362.889} C_VEL
LIN {X 0,Y 63.914,Z 303.136,A -85,B 0,C 180,E1 -28369.264,E2 -28369.264} C_VEL
LIN {X 0,Y 65.498,Z 303.352,A -85,B 0,C 180,E1 -28375.419,E2 -28375.419} C_VEL
LIN {X 0,Y 70.709,Z 302.534,A -85,B 0,C 180,E1 -28386.612,E2 -28386.612} C_VEL
LIN {X 0,Y 74.101,Z 301.544,A -85,B 0,C 180,E1 -28391.601,E2 -28391.601} C_VEL
LIN {X 0,Y 77.927,Z 300.123,A -85,B 0,C 180,E1 -28396.181,E2 -28396.181} C_VEL
LIN {X 0,Y 84.479,Z 297.17,A -85,B 0,C 180,E1 -28402.218,E2 -28402.218} C_VEL
LIN {X 0,Y 93.018,Z 292.397,A -85,B 0,C 180,E1 -28408.068,E2 -28408.068} C_VEL
LIN {X 0,Y 102.565,Z 285.906,A -85,B 0,C 180,E1 -28412.975,E2 -28412.975} C_VEL
LIN {X 0,Y 111.142,Z 278.809,A -85,B 0,C 180,E1 -28416.48,E2 -28416.48} C_VEL
LIN {X 0,Y 119.982,Z 269.916,A -85,B 0,C 180,E1 -28419.59,E2 -28419.59} C_VEL
LIN {X 0,Y 127.611,Z 260.76,A -85,B 0,C 180,E1 -28421.812,E2 -28421.812} C_VEL
LIN {X 0,Y 134.644,Z 250.558,A -85,B 0,C 180,E1 -28423.563,E2 -28423.563} C_VEL
LIN {X 0,Y 141.001,Z 239.185,A -85,B 0,C 180,E1 -28424.958,E2 -28424.958} C_VEL
LIN {X 0,Y 145.803,Z 228.186,A -85,B 0,C 180,E1 -28426.053,E2 -28426.053} C_VEL
LIN {X 0,Y 149.768,Z 216.512,A -85,B 0,C 180,E1 -28426.822,E2 -28426.822} C_VEL
LIN {X 0,Y 152.568,Z 204.757,A -85,B 0,C 180,E1 -28427.392,E2 -28427.392} C_VEL
LIN {X 0,Y 151.013,Z 199.762,A -85,B 0,C 180,E1 -28431.3,E2 -28431.3} C_VEL
LIN {X 0,Y 150.085,Z 197.256,A -85,B 0,C 180,E1 -28433.951,E2 -28433.951} C_VEL
LIN {X 0,Y 149.093,Z 194.181,A -85,B 0,C 180,E1 -28438.311,E2 -28438.311} C_VEL
LIN {X 0,Y 148.618,Z 193.563,A -85,B 0,C 180,E1 -28442.71,E2 -28442.71} C_VEL
LIN {X 0,Y 149.119,Z 194.401,A -85,B 0,C 180,E1 -28448.341,E2 -28448.341} C_VEL
LIN {X 0,Y 150.46,Z 198.263,A -85,B 0,C 180,E1 -28453.506,E2 -28453.506} C_VEL
LIN {X 0,Y 151.087,Z 200.538,A -85,B 0,C 180,E1 -28455.34,E2 -28455.34} C_VEL
LIN {X 0,Y 152.119,Z 205.799,A -85,B 0,C 180,E1 -28458.345,E2 -28458.345} C_VEL
LIN {X 0,Y 152.329,Z 207.256,A -85,B 0,C 180,E1 -28459.016,E2 -28459.016} C_VEL
LIN {X 0,Y 149.656,Z 218.896,A -85,B 0,C 180,E1 -28459.502,E2 -28459.502} C_VEL
LIN {X 0,Y 145.463,Z 231.548,A -85,B 0,C 180,E1 -28460.258,E2 -28460.258} C_VEL
LIN {X 0,Y 140.352,Z 242.961,A -85,B 0,C 180,E1 -28461.148,E2 -28461.148} C_VEL
LIN {X 0,Y 133.975,Z 254.284,A -85,B 0,C 180,E1 -28462.395,E2 -28462.395} C_VEL
LIN {X 0,Y 126.851,Z 264.512,A -85,B 0,C 180,E1 -28463.911,E2 -28463.911} C_VEL
LIN {X 0,Y 119.189,Z 273.708,A -85,B 0,C 180,E1 -28465.942,E2 -28465.942} C_VEL
LIN {X 0,Y 111.649,Z 281.316,A -85,B 0,C 180,E1 -28468.203,E2 -28468.203} C_VEL
LIN {X 0,Y 102.94,Z 288.79,A -85,B 0,C 180,E1 -28471.413,E2 -28471.413} C_VEL
LIN {X 0,Y 94.674,Z 294.817,A -85,B 0,C 180,E1 -28475.255,E2 -28475.255} C_VEL
LIN {X 0,Y 87.017,Z 299.609,A -85,B 0,C 180,E1 -28479.888,E2 -28479.888} C_VEL
LIN {X 0,Y 80.044,Z 303.305,A -85,B 0,C 180,E1 -28485.377,E2 -28485.377} C_VEL
LIN {X 0,Y 75.807,Z 305.229,A -85,B 0,C 180,E1 -28489.534,E2 -28489.534} C_VEL
LIN {X 0,Y 72.085,Z 306.714,A -85,B 0,C 180,E1 -28494.196,E2 -28494.196} C_VEL
LIN {X 0,Y 66.255,Z 308.47,A -85,B 0,C 180,E1 -28504.892,E2 -28504.892} C_VEL
LIN {X 0,Y 64.408,Z 308.783,A -85,B 0,C 180,E1 -28510.89,E2 -28510.89} C_VEL
LIN {X 0,Y 63.224,Z 308.696,A -85,B 0,C 180,E1 -28517.153,E2 -28517.153} C_VEL
LIN {X 0,Y 62.745,Z 308.19,A -85,B 0,C 180,E1 -28523.567,E2 -28523.567} C_VEL
LIN {X 0,Y 62.85,Z 307.292,A -85,B 0,C 180,E1 -28529.998,E2 -28529.998} C_VEL
LIN {X 0,Y 62.735,Z 305.947,A -85,B 0,C 180,E1 -28536.43,E2 -28536.43} C_VEL
LIN {X 0,Y 63.657,Z 303.075,A -85,B 0,C 180,E1 -28546.02,E2 -28546.02} C_VEL
LIN {X 0,Y 66.045,Z 299.149,A -85,B 0,C 180,E1 -28555.19,E2 -28555.19} C_VEL
LIN {X 0,Y 70.089,Z 294.092,A -85,B 0,C 180,E1 -28563.468,E2 -28563.468} C_VEL
LIN {X 0,Y 75.36,Z 287.729,A -85,B 0,C 180,E1 -28570.752,E2 -28570.752} C_VEL
LIN {X 0,Y 80.398,Z 281.199,A -85,B 0,C 180,E1 -28576.149,E2 -28576.149} C_VEL
LIN {X 0,Y 86.163,Z 273.367,A -85,B 0,C 180,E1 -28580.792,E2 -28580.792} C_VEL
LIN {X 0,Y 92.501,Z 263.807,A -85,B 0,C 180,E1 -28584.759,E2 -28584.759} C_VEL
LIN {X 0,Y 98.564,Z 253.2,A -85,B 0,C 180,E1 -28587.856,E2 -28587.856} C_VEL
LIN {X 0,Y 104.21,Z 241.369,A -85,B 0,C 180,E1 -28590.259,E2 -28590.259} C_VEL
LIN {X 0,Y 108.928,Z 228.67,A -85,B 0,C 180,E1 -28592.018,E2 -28592.018} C_VEL
LIN {X 0,Y 112.389,Z 215.626,A -85,B 0,C 180,E1 -28593.35,E2 -28593.35} C_VEL
LIN {X 0,Y 114.674,Z 202.454,A -85,B 0,C 180,E1 -28594.153,E2 -28594.153} C_VEL
LIN {X 0,Y 117.252,Z 176.542,A -85,B 0,C 180,E1 -28595.193,E2 -28595.193} C_VEL
LIN {X 0,Y 115.089,Z 168.633,A -85,B 0,C 180,E1 -28598.346,E2 -28598.346} C_VEL
LIN {X 0,Y 112.309,Z 162.7,A -85,B 0,C 180,E1 -28602.518,E2 -28602.518} C_VEL
LIN {X 0,Y 110.27,Z 158.754,A -85,B 0,C 180,E1 -28606.247,E2 -28606.247} C_VEL
LIN {X 0,Y 108.537,Z 155.481,A -85,B 0,C 180,E1 -28610.303,E2 -28610.303} C_VEL
LIN {X 0,Y 107.004,Z 152.144,A -85,B 0,C 180,E1 -28615.749,E2 -28615.749} C_VEL
LIN {X 0,Y 106.735,Z 151.565,A -85,B 0,C 180,E1 -28617.17,E2 -28617.17} C_VEL
LIN {X 0,Y 106.315,Z 151.073,A -85,B 0,C 180,E1 -28620.001,E2 -28620.001} C_VEL
LIN {X 0,Y 106.387,Z 151.457,A -85,B 0,C 180,E1 -28628.549,E2 -28628.549} C_VEL
LIN {X 0,Y 106.592,Z 151.621,A -85,B 0,C 180,E1 -28629.852,E2 -28629.852} C_VEL
LIN {X 0,Y 106.963,Z 152.373,A -85,B 0,C 180,E1 -28631.891,E2 -28631.891} C_VEL
LIN {X 0,Y 107.52,Z 154.912,A -85,B 0,C 180,E1 -28634.712,E2 -28634.712} C_VEL
LIN {X 0,Y 108.089,Z 158.463,A -85,B 0,C 180,E1 -28637.238,E2 -28637.238} C_VEL
LIN {X 0,Y 109.633,Z 166.684,A -85,B 0,C 180,E1 -28642.081,E2 -28642.081} C_VEL
LIN {X 0,Y 110.435,Z 169.114,A -85,B 0,C 180,E1 -28643.771,E2 -28643.771} C_VEL
LIN {X 0,Y 113.05,Z 175.202,A -85,B 0,C 180,E1 -28648.108,E2 -28648.108} C_VEL
LIN {X 0,Y 113.845,Z 177.3,A -85,B 0,C 180,E1 -28649.288,E2 -28649.288} C_VEL
LIN {X 0,Y 111.256,Z 201.28,A -85,B 0,C 180,E1 -28650.325,E2 -28650.325} C_VEL
LIN {X 0,Y 108.498,Z 215.025,A -85,B 0,C 180,E1 -28651.363,E2 -28651.363} C_VEL
LIN {X 0,Y 105.007,Z 226.958,A -85,B 0,C 180,E1 -28652.778,E2 -28652.778} C_VEL
LIN {X 0,Y 100.467,Z 238.64,A -85,B 0,C 180,E1 -28654.721,E2 -28654.721} C_VEL
LIN {X 0,Y 94.874,Z 249.925,A -85,B 0,C 180,E1 -28657.221,E2 -28657.221} C_VEL
LIN {X 0,Y 88.798,Z 260.103,A -85,B 0,C 180,E1 -28660.381,E2 -28660.381} C_VEL
LIN {X 0,Y 81.691,Z 270.066,A -85,B 0,C 180,E1 -28664.786,E2 -28664.786} C_VEL
LIN {X 0,Y 74.593,Z 278.827,A -85,B 0,C 180,E1 -28670.51,E2 -28670.51} C_VEL
LIN {X 0,Y 68.262,Z 285.85,A -85,B 0,C 180,E1 -28677.283,E2 -28677.283} C_VEL
LIN {X 0,Y 62.296,Z 292.255,A -85,B 0,C 180,E1 -28686.745,E2 -28686.745} C_VEL
LIN {X 0,Y 58.662,Z 296.485,A -85,B 0,C 180,E1 -28696.139,E2 -28696.139} C_VEL
LIN {X 0,Y 56.246,Z 300.18,A -85,B 0,C 180,E1 -28708.453,E2 -28708.453} C_VEL
LIN {X 0,Y 55.697,Z 301.907,A -85,B 0,C 180,E1 -28717.251,E2 -28717.251} C_VEL
LIN {X 0,Y 56.055,Z 302.891,A -85,B 0,C 180,E1 -28724.524,E2 -28724.524} C_VEL
LIN {X 0,Y 57.186,Z 303.491,A -85,B 0,C 180,E1 -28731.637,E2 -28731.637} C_VEL
LIN {X 0,Y 59.102,Z 303.665,A -85,B 0,C 180,E1 -28738.404,E2 -28738.404} C_VEL
LIN {X 0,Y 65.079,Z 302.807,A -85,B 0,C 180,E1 -28750.39,E2 -28750.39} C_VEL
LIN {X 0,Y 68.869,Z 301.797,A -85,B 0,C 180,E1 -28755.592,E2 -28755.592} C_VEL
LIN {X 0,Y 73.112,Z 300.335,A -85,B 0,C 180,E1 -28760.268,E2 -28760.268} C_VEL
LIN {X 0,Y 80.262,Z 297.337,A -85,B 0,C 180,E1 -28766.292,E2 -28766.292} C_VEL
LIN {X 0,Y 88.713,Z 292.925,A -85,B 0,C 180,E1 -28771.618,E2 -28771.618} C_VEL
LIN {X 0,Y 98.044,Z 286.982,A -85,B 0,C 180,E1 -28776.06,E2 -28776.06} C_VEL
LIN {X 0,Y 106.958,Z 280.111,A -85,B 0,C 180,E1 -28779.449,E2 -28779.449} C_VEL
LIN {X 0,Y 115.75,Z 271.84,A -85,B 0,C 180,E1 -28782.326,E2 -28782.326} C_VEL
LIN {X 0,Y 123.965,Z 262.551,A -85,B 0,C 180,E1 -28784.538,E2 -28784.538} C_VEL
LIN {X 0,Y 131.181,Z 252.729,A -85,B 0,C 180,E1 -28786.182,E2 -28786.182} C_VEL
LIN {X 0,Y 137.627,Z 242.004,A -85,B 0,C 180,E1 -28787.474,E2 -28787.474} C_VEL
LIN {X 0,Y 143.368,Z 229.651,A -85,B 0,C 180,E1 -28788.647,E2 -28788.647} C_VEL
LIN {X 0,Y 147.808,Z 217.059,A -85,B 0,C 180,E1 -28789.442,E2 -28789.442} C_VEL
LIN {X 0,Y 149.883,Z 208.989,A -85,B 0,C 180,E1 -28789.846,E2 -28789.846} C_VEL
LIN {X 0,Y 148.989,Z 205.235,A -85,B 0,C 180,E1 -28793.227,E2 -28793.227} C_VEL
LIN {X 0,Y 148.346,Z 203.164,A -85,B 0,C 180,E1 -28795.924,E2 -28795.924} C_VEL
LIN {X 0,Y 147.993,Z 201.109,A -85,B 0,C 180,E1 -28798.809,E2 -28798.809} C_VEL
LIN {X 0,Y 147.65,Z 200.582,A -85,B 0,C 180,E1 -28802.728,E2 -28802.728} C_VEL
LIN {X 0,Y 148.045,Z 201.373,A -85,B 0,C 180,E1 -28807.879,E2 -28807.879} C_VEL
LIN {X 0,Y 148.972,Z 204.792,A -85,B 0,C 180,E1 -28812.602,E2 -28812.602} C_VEL
LIN {X 0,Y 149.455,Z 207.414,A -85,B 0,C 180,E1 -28814.64,E2 -28814.64} C_VEL
LIN {X 0,Y 149.814,Z 210.662,A -85,B 0,C 180,E1 -28816.522,E2 -28816.522} C_VEL
LIN {X 0,Y 146.641,Z 222.563,A -85,B 0,C 180,E1 -28817.044,E2 -28817.044} C_VEL
LIN {X 0,Y 142.034,Z 234.907,A -85,B 0,C 180,E1 -28817.76,E2 -28817.76} C_VEL
LIN {X 0,Y 136.323,Z 246.478,A -85,B 0,C 180,E1 -28818.68,E2 -28818.68} C_VEL
LIN {X 0,Y 128.982,Z 258.171,A -85,B 0,C 180,E1 -28819.959,E2 -28819.959} C_VEL
LIN {X 0,Y 122.564,Z 266.626,A -85,B 0,C 180,E1 -28821.28,E2 -28821.28} C_VEL
LIN {X 0,Y 114.664,Z 275.414,A -85,B 0,C 180,E1 -28823.161,E2 -28823.161} C_VEL
LIN {X 0,Y 105.443,Z 283.996,A -85,B 0,C 180,E1 -28825.864,E2 -28825.864} C_VEL
LIN {X 0,Y 96.476,Z 290.881,A -85,B 0,C 180,E1 -28829.051,E2 -28829.051} C_VEL
LIN {X 0,Y 87.964,Z 296.419,A -85,B 0,C 180,E1 -28832.972,E2 -28832.972} C_VEL
LIN {X 0,Y 79.185,Z 301.218,A -85,B 0,C 180,E1 -28838.408,E2 -28838.408} C_VEL
LIN {X 0,Y 70.541,Z 305.012,A -85,B 0,C 180,E1 -28845.778,E2 -28845.778} C_VEL
LIN {X 0,Y 66.444,Z 306.46,A -85,B 0,C 180,E1 -28850.604,E2 -28850.604} C_VEL
LIN {X 0,Y 59.863,Z 308.176,A -85,B 0,C 180,E1 -28861.989,E2 -28861.989} C_VEL
LIN {X 0,Y 57.715,Z 308.47,A -85,B 0,C 180,E1 -28868.571,E2 -28868.571} C_VEL
LIN {X 0,Y 56.297,Z 308.346,A -85,B 0,C 180,E1 -28875.539,E2 -28875.539} C_VEL
LIN {X 0,Y 55.672,Z 307.821,A -85,B 0,C 180,E1 -28882.746,E2 -28882.746} C_VEL
LIN {X 0,Y 55.754,Z 306.904,A -85,B 0,C 180,E1 -28889.998,E2 -28889.998} C_VEL
LIN {X 0,Y 55.65,Z 305.538,A -85,B 0,C 180,E1 -28897.253,E2 -28897.253} C_VEL
LIN {X 0,Y 56.808,Z 302.623,A -85,B 0,C 180,E1 -28908.014,E2 -28908.014} C_VEL
LIN {X 0,Y 59.654,Z 298.655,A -85,B 0,C 180,E1 -28918.113,E2 -28918.113} C_VEL
LIN {X 0,Y 65.102,Z 292.559,A -85,B 0,C 180,E1 -28928.368,E2 -28928.368} C_VEL
LIN {X 0,Y 70.048,Z 287.113,A -85,B 0,C 180,E1 -28934.611,E2 -28934.611} C_VEL
LIN {X 0,Y 76.814,Z 279.042,A -85,B 0,C 180,E1 -28941.048,E2 -28941.048} C_VEL
LIN {X 0,Y 83.141,Z 270.826,A -85,B 0,C 180,E1 -28945.502,E2 -28945.502} C_VEL
LIN {X 0,Y 90.024,Z 260.825,A -85,B 0,C 180,E1 -28949.174,E2 -28949.174} C_VEL
LIN {X 0,Y 96.403,Z 249.501,A -85,B 0,C 180,E1 -28952.119,E2 -28952.119} C_VEL
LIN {X 0,Y 101.606,Z 238.418,A -85,B 0,C 180,E1 -28954.051,E2 -28954.051} C_VEL
LIN {X 0,Y 106.138,Z 226.113,A -85,B 0,C 180,E1 -28955.567,E2 -28955.567} C_VEL
LIN {X 0,Y 109.513,Z 213.086,A -85,B 0,C 180,E1 -28956.7,E2 -28956.7} C_VEL
LIN {X 0,Y 111.574,Z 200.558,A -85,B 0,C 180,E1 -28957.4,E2 -28957.4} C_VEL
LIN {X 0,Y 113.779,Z 178.931,A -85,B 0,C 180,E1 -28958.247,E2 -28958.247} C_VEL
LIN {X 0,Y 112.36,Z 173.427,A -85,B 0,C 180,E1 -28960.671,E2 -28960.671} C_VEL
LIN {X 0,Y 109.685,Z 167.322,A -85,B 0,C 180,E1 -28965.406,E2 -28965.406} C_VEL
LIN {X 0,Y 108.227,Z 164.369,A -85,B 0,C 180,E1 -28968.607,E2 -28968.607} C_VEL
LIN {X 0,Y 107.19,Z 162.091,A -85,B 0,C 180,E1 -28971.488,E2 -28971.488} C_VEL
LIN {X 0,Y 105.861,Z 158.652,A -85,B 0,C 180,E1 -28977.147,E2 -28977.147} C_VEL
LIN {X 0,Y 105.419,Z 158.108,A -85,B 0,C 180,E1 -28980.238,E2 -28980.238} C_VEL
LIN {X 0,Y 105.528,Z 158.502,A -85,B 0,C 180,E1 -28988.619,E2 -28988.619} C_VEL
LIN {X 0,Y 105.815,Z 158.995,A -85,B 0,C 180,E1 -28990.525,E2 -28990.525} C_VEL
LIN {X 0,Y 107.657,Z 163.215,A -85,B 0,C 180,E1 -28997.615,E2 -28997.615} C_VEL
LIN {X 0,Y 109.577,Z 167.258,A -85,B 0,C 180,E1 -29002.111,E2 -29002.111} C_VEL
LIN {X 0,Y 110.435,Z 169.114,A -85,B 0,C 180,E1 -29003.771,E2 -29003.771} C_VEL
LIN {X 0,Y 111.082,Z 171.78,A -85,B 0,C 180,E1 -29005.121,E2 -29005.121} C_VEL
LIN {X 0,Y 111.366,Z 175.185,A -85,B 0,C 180,E1 -29006.021,E2 -29006.021} C_VEL
LIN {X 0,Y 111.23,Z 180.972,A -85,B 0,C 180,E1 -29006.727,E2 -29006.727} C_VEL
LIN {X 0,Y 109.891,Z 191.634,A -85,B 0,C 180,E1 -29006.843,E2 -29006.843} C_VEL
LIN {X 0,Y 108.477,Z 200.283,A -85,B 0,C 180,E1 -29006.912,E2 -29006.912} C_VEL
LIN {X 0,Y 105.769,Z 213.769,A -85,B 0,C 180,E1 -29007.817,E2 -29007.817} C_VEL
LIN {X 0,Y 102.111,Z 226.234,A -85,B 0,C 180,E1 -29009.164,E2 -29009.164} C_VEL
LIN {X 0,Y 97.356,Z 238.18,A -85,B 0,C 180,E1 -29010.994,E2 -29010.994} C_VEL
LIN {X 0,Y 91.499,Z 249.607,A -85,B 0,C 180,E1 -29013.354,E2 -29013.354} C_VEL
LIN {X 0,Y 85.099,Z 259.904,A -85,B 0,C 180,E1 -29016.371,E2 -29016.371} C_VEL
LIN {X 0,Y 78.202,Z 269.174,A -85,B 0,C 180,E1 -29020.193,E2 -29020.193} C_VEL
LIN {X 0,Y 70.485,Z 278.14,A -85,B 0,C 180,E1 -29025.738,E2 -29025.738} C_VEL
LIN {X 0,Y 63.498,Z 285.369,A -85,B 0,C 180,E1 -29032.504,E2 -29032.504} C_VEL
LIN {X 0,Y 57.551,Z 291.156,A -85,B 0,C 180,E1 -29040.762,E2 -29040.762} C_VEL
LIN {X 0,Y 53.016,Z 295.709,A -85,B 0,C 180,E1 -29050.648,E2 -29050.648} C_VEL
LIN {X 0,Y 49.955,Z 299.193,A -85,B 0,C 180,E1 -29061.915,E2 -29061.915} C_VEL
LIN {X 0,Y 48.953,Z 300.949,A -85,B 0,C 180,E1 -29070.002,E2 -29070.002} C_VEL
LIN {X 0,Y 48.609,Z 302.302,A -85,B 0,C 180,E1 -29078.316,E2 -29078.316} C_VEL
LIN {X 0,Y 49.158,Z 303.265,A -85,B 0,C 180,E1 -29086.617,E2 -29086.617} C_VEL
LIN {X 0,Y 50.572,Z 303.841,A -85,B 0,C 180,E1 -29094.642,E2 -29094.642} C_VEL
LIN {X 0,Y 56.009,Z 303.723,A -85,B 0,C 180,E1 -29108.862,E2 -29108.862} C_VEL
LIN {X 0,Y 60.394,Z 302.963,A -85,B 0,C 180,E1 -29115.714,E2 -29115.714} C_VEL
LIN {X 0,Y 68.731,Z 300.546,A -85,B 0,C 180,E1 -29124.891,E2 -29124.891} C_VEL
LIN {X 0,Y 76.501,Z 297.504,A -85,B 0,C 180,E1 -29130.783,E2 -29130.783} C_VEL
LIN {X 0,Y 84.922,Z 293.383,A -85,B 0,C 180,E1 -29135.556,E2 -29135.556} C_VEL
LIN {X 0,Y 95.352,Z 287.05,A -85,B 0,C 180,E1 -29140.014,E2 -29140.014} C_VEL
LIN {X 0,Y 104.647,Z 280.116,A -85,B 0,C 180,E1 -29143.145,E2 -29143.145} C_VEL
LIN {X 0,Y 113.801,Z 271.718,A -85,B 0,C 180,E1 -29145.793,E2 -29145.793} C_VEL
LIN {X 0,Y 122.244,Z 262.377,A -85,B 0,C 180,E1 -29147.789,E2 -29147.789} C_VEL
LIN {X 0,Y 129.654,Z 252.455,A -85,B 0,C 180,E1 -29149.264,E2 -29149.264} C_VEL
LIN {X 0,Y 136.175,Z 241.666,A -85,B 0,C 180,E1 -29150.412,E2 -29150.412} C_VEL
LIN {X 0,Y 142.125,Z 228.959,A -85,B 0,C 180,E1 -29151.495,E2 -29151.495} C_VEL
LIN {X 0,Y 146.213,Z 217.466,A -85,B 0,C 180,E1 -29152.127,E2 -29152.127} C_VEL
LIN {X 0,Y 147.315,Z 213.423,A -85,B 0,C 180,E1 -29152.375,E2 -29152.375} C_VEL
LIN {X 0,Y 146.844,Z 210.489,A -85,B 0,C 180,E1 -29155.539,E2 -29155.539} C_VEL
LIN {X 0,Y 146.518,Z 207.957,A -85,B 0,C 180,E1 -29159.312,E2 -29159.312} C_VEL
LIN {X 0,Y 146.323,Z 207.538,A -85,B 0,C 180,E1 -29162.752,E2 -29162.752} C_VEL
LIN {X 0,Y 146.622,Z 208.36,A -85,B 0,C 180,E1 -29167.574,E2 -29167.574} C_VEL
LIN {X 0,Y 147.24,Z 211.603,A -85,B 0,C 180,E1 -29172.053,E2 -29172.053} C_VEL
LIN {X 0,Y 147.444,Z 214.282,A -85,B 0,C 180,E1 -29173.963,E2 -29173.963} C_VEL
LIN {X 0,Y 143.702,Z 226.446,A -85,B 0,C 180,E1 -29174.515,E2 -29174.515} C_VEL
LIN {X 0,Y 138.39,Z 238.991,A -85,B 0,C 180,E1 -29175.223,E2 -29175.223} C_VEL
LIN {X 0,Y 132.561,Z 249.702,A -85,B 0,C 180,E1 -29176.064,E2 -29176.064} C_VEL
LIN {X 0,Y 125.915,Z 259.578,A -85,B 0,C 180,E1 -29177.087,E2 -29177.087} C_VEL
LIN {X 0,Y 118.548,Z 268.676,A -85,B 0,C 180,E1 -29178.457,E2 -29178.457} C_VEL
LIN {X 0,Y 110.466,Z 277.027,A -85,B 0,C 180,E1 -29180.209,E2 -29180.209} C_VEL
LIN {X 0,Y 100.973,Z 285.211,A -85,B 0,C 180,E1 -29182.742,E2 -29182.742} C_VEL
LIN {X 0,Y 93.236,Z 290.807,A -85,B 0,C 180,E1 -29185.235,E2 -29185.235} C_VEL
LIN {X 0,Y 84.307,Z 296.295,A -85,B 0,C 180,E1 -29188.916,E2 -29188.916} C_VEL
LIN {X 0,Y 74.166,Z 301.419,A -85,B 0,C 180,E1 -29194.649,E2 -29194.649} C_VEL
LIN {X 0,Y 65.627,Z 304.789,A -85,B 0,C 180,E1 -29201.438,E2 -29201.438} C_VEL
LIN {X 0,Y 57.057,Z 307.234,A -85,B 0,C 180,E1 -29211.982,E2 -29211.982} C_VEL
LIN {X 0,Y 51.128,Z 308.151,A -85,B 0,C 180,E1 -29225.643,E2 -29225.643} C_VEL
LIN {X 0,Y 49.439,Z 307.995,A -85,B 0,C 180,E1 -29233.48,E2 -29233.48} C_VEL
LIN {X 0,Y 48.616,Z 307.451,A -85,B 0,C 180,E1 -29241.686,E2 -29241.686} C_VEL
LIN {X 0,Y 48.648,Z 306.516,A -85,B 0,C 180,E1 -29249.998,E2 -29249.998} C_VEL
LIN {X 0,Y 48.596,Z 305.126,A -85,B 0,C 180,E1 -29258.313,E2 -29258.313} C_VEL
LIN {X 0,Y 50.05,Z 302.171,A -85,B 0,C 180,E1 -29270.549,E2 -29270.549} C_VEL
LIN {X 0,Y 53.457,Z 298.16,A -85,B 0,C 180,E1 -29281.725,E2 -29281.725} C_VEL
LIN {X 0,Y 59.645,Z 291.989,A -85,B 0,C 180,E1 -29292.648,E2 -29292.648} C_VEL
LIN {X 0,Y 65.079,Z 286.48,A -85,B 0,C 180,E1 -29299.105,E2 -29299.105} C_VEL
LIN {X 0,Y 72.522,Z 278.352,A -85,B 0,C 180,E1 -29305.456,E2 -29305.456} C_VEL
LIN {X 0,Y 79.309,Z 270.064,A -85,B 0,C 180,E1 -29309.765,E2 -29309.765} C_VEL
LIN {X 0,Y 86.563,Z 259.958,A -85,B 0,C 180,E1 -29313.261,E2 -29313.261} C_VEL
LIN {X 0,Y 92.522,Z 249.914,A -85,B 0,C 180,E1 -29315.713,E2 -29315.713} C_VEL
LIN {X 0,Y 97.919,Z 239.005,A -85,B 0,C 180,E1 -29317.528,E2 -29317.528} C_VEL
LIN {X 0,Y 102.611,Z 226.955,A -85,B 0,C 180,E1 -29318.935,E2 -29318.935} C_VEL
LIN {X 0,Y 106.154,Z 214.302,A -85,B 0,C 180,E1 -29320.042,E2 -29320.042} C_VEL
LIN {X 0,Y 108.461,Z 201.572,A -85,B 0,C 180,E1 -29320.723,E2 -29320.723} C_VEL
LIN {X 0,Y 110.625,Z 181.491,A -85,B 0,C 180,E1 -29321.48,E2 -29321.48} C_VEL
LIN {X 0,Y 109.904,Z 178.574,A -85,B 0,C 180,E1 -29322.933,E2 -29322.933} C_VEL
LIN {X 0,Y 107.83,Z 173.29,A -85,B 0,C 180,E1 -29327.218,E2 -29327.218} C_VEL
LIN {X 0,Y 106.551,Z 170.356,A -85,B 0,C 180,E1 -29330.532,E2 -29330.532} C_VEL
LIN {X 0,Y 105.773,Z 168.56,A -85,B 0,C 180,E1 -29333.084,E2 -29333.084} C_VEL
LIN {X 0,Y 104.821,Z 165.55,A -85,B 0,C 180,E1 -29338.08,E2 -29338.08} C_VEL
LIN {X 0,Y 104.348,Z 165.139,A -85,B 0,C 180,E1 -29343.863,E2 -29343.863} C_VEL
LIN {X 0,Y 104.784,Z 165.828,A -85,B 0,C 180,E1 -29349.593,E2 -29349.593} C_VEL
LIN {X 0,Y 106.351,Z 169.944,A -85,B 0,C 180,E1 -29356.575,E2 -29356.575} C_VEL
LIN {X 0,Y 108.208,Z 174.25,A -85,B 0,C 180,E1 -29361.351,E2 -29361.351} C_VEL
LIN {X 0,Y 110.562,Z 180.446,A -85,B 0,C 180,E1 -29365.966,E2 -29365.966} C_VEL
LIN {X 0,Y 110.652,Z 180.701,A -85,B 0,C 180,E1 -29366.124,E2 -29366.124} C_VEL
LIN {X 0,Y 108.477,Z 200.283,A -85,B 0,C 180,E1 -29366.912,E2 -29366.912} C_VEL
LIN {X 0,Y 107.199,Z 206.061,A -85,B 0,C 180,E1 -29366.878,E2 -29366.878} C_VEL
LIN {X 0,Y 102.513,Z 218.988,A -85,B 0,C 180,E1 -29365.819,E2 -29365.819} C_VEL
LIN {X 0,Y 99.457,Z 226.286,A -85,B 0,C 180,E1 -29365.606,E2 -29365.606} C_VEL
LIN {X 0,Y 98.004,Z 229.869,A -85,B 0,C 180,E1 -29365.904,E2 -29365.904} C_VEL
LIN {X 0,Y 92.38,Z 242.419,A -85,B 0,C 180,E1 -29367.825,E2 -29367.825} C_VEL
LIN {X 0,Y 85.565,Z 254.185,A -85,B 0,C 180,E1 -29370.412,E2 -29370.412} C_VEL
LIN {X 0,Y 78.136,Z 264.648,A -85,B 0,C 180,E1 -29373.699,E2 -29373.699} C_VEL
LIN {X 0,Y 71.031,Z 273.111,A -85,B 0,C 180,E1 -29377.673,E2 -29377.673} C_VEL
LIN {X 0,Y 62.992,Z 281.353,A -85,B 0,C 180,E1 -29383.517,E2 -29383.517} C_VEL
LIN {X 0,Y 55.735,Z 287.997,A -85,B 0,C 180,E1 -29390.917,E2 -29390.917} C_VEL
LIN {X 0,Y 49.621,Z 293.297,A -85,B 0,C 180,E1 -29400.286,E2 -29400.286} C_VEL
LIN {X 0,Y 45.03,Z 297.437,A -85,B 0,C 180,E1 -29411.814,E2 -29411.814} C_VEL
LIN {X 0,Y 42.346,Z 300.449,A -85,B 0,C 180,E1 -29424.766,E2 -29424.766} C_VEL
LIN {X 0,Y 41.542,Z 302.696,A -85,B 0,C 180,E1 -29439.743,E2 -29439.743} C_VEL
LIN {X 0,Y 42.327,Z 303.641,A -85,B 0,C 180,E1 -29449.398,E2 -29449.398} C_VEL
LIN {X 0,Y 44.143,Z 304.183,A -85,B 0,C 180,E1 -29458.534,E2 -29458.534} C_VEL
LIN {X 0,Y 50.608,Z 304.017,A -85,B 0,C 180,E1 -29473.98,E2 -29473.98} C_VEL
LIN {X 0,Y 55.03,Z 303.335,A -85,B 0,C 180,E1 -29480.313,E2 -29480.313} C_VEL
LIN {X 0,Y 59.66,Z 302.281,A -85,B 0,C 180,E1 -29485.552,E2 -29485.552} C_VEL
LIN {X 0,Y 64.842,Z 300.758,A -85,B 0,C 180,E1 -29490.126,E2 -29490.126} C_VEL
LIN {X 0,Y 73.26,Z 297.671,A -85,B 0,C 180,E1 -29495.697,E2 -29495.697} C_VEL
LIN {X 0,Y 82.206,Z 293.502,A -85,B 0,C 180,E1 -29500.127,E2 -29500.127} C_VEL
LIN {X 0,Y 93.133,Z 287.118,A -85,B 0,C 180,E1 -29504.189,E2 -29504.189} C_VEL
LIN {X 0,Y 102.79,Z 280.105,A -85,B 0,C 180,E1 -29506.989,E2 -29506.989} C_VEL
LIN {X 0,Y 111.92,Z 271.96,A -85,B 0,C 180,E1 -29509.271,E2 -29509.271} C_VEL
LIN {X 0,Y 120.922,Z 262.203,A -85,B 0,C 180,E1 -29511.137,E2 -29511.137} C_VEL
LIN {X 0,Y 128.51,Z 252.156,A -85,B 0,C 180,E1 -29512.411,E2 -29512.411} C_VEL
LIN {X 0,Y 135.732,Z 240.116,A -85,B 0,C 180,E1 -29513.502,E2 -29513.502} C_VEL
LIN {X 0,Y 141.244,Z 228.271,A -85,B 0,C 180,E1 -29514.368,E2 -29514.368} C_VEL
LIN {X 0,Y 144.314,Z 219.804,A -85,B 0,C 180,E1 -29514.786,E2 -29514.786} C_VEL
LIN {X 0,Y 144.843,Z 217.977,A -85,B 0,C 180,E1 -29515.058,E2 -29515.058} C_VEL
LIN {X 0,Y 144.673,Z 214.711,A -85,B 0,C 180,E1 -29519.999,E2 -29519.999} C_VEL
LIN {X 0,Y 144.576,Z 214.433,A -85,B 0,C 180,E1 -29522.786,E2 -29522.786} C_VEL
LIN {X 0,Y 144.799,Z 215.149,A -85,B 0,C 180,E1 -29527.144,E2 -29527.144} C_VEL
LIN {X 0,Y 145.126,Z 217.977,A -85,B 0,C 180,E1 -29531.169,E2 -29531.169} C_VEL
LIN {X 0,Y 144.767,Z 219.473,A -85,B 0,C 180,E1 -29531.433,E2 -29531.433} C_VEL
LIN {X 0,Y 140.033,Z 232.358,A -85,B 0,C 180,E1 -29532.007,E2 -29532.007} C_VEL
LIN {X 0,Y 134.156,Z 244.319,A -85,B 0,C 180,E1 -29532.652,E2 -29532.652} C_VEL
LIN {X 0,Y 127.41,Z 255.154,A -85,B 0,C 180,E1 -29533.536,E2 -29533.536} C_VEL
LIN {X 0,Y 119.821,Z 264.988,A -85,B 0,C 180,E1 -29534.576,E2 -29534.576} C_VEL
LIN {X 0,Y 111.522,Z 273.939,A -85,B 0,C 180,E1 -29536.043,E2 -29536.043} C_VEL
LIN {X 0,Y 101.679,Z 282.702,A -85,B 0,C 180,E1 -29538.119,E2 -29538.119} C_VEL
LIN {X 0,Y 92.016,Z 289.719,A -85,B 0,C 180,E1 -29540.666,E2 -29540.666} C_VEL
LIN {X 0,Y 81.104,Z 296.17,A -85,B 0,C 180,E1 -29544.509,E2 -29544.509} C_VEL
LIN {X 0,Y 72.198,Z 300.447,A -85,B 0,C 180,E1 -29548.823,E2 -29548.823} C_VEL
LIN {X 0,Y 66.524,Z 302.728,A -85,B 0,C 180,E1 -29552.307,E2 -29552.307} C_VEL
LIN {X 0,Y 61.149,Z 304.558,A -85,B 0,C 180,E1 -29556.432,E2 -29556.432} C_VEL
LIN {X 0,Y 51.644,Z 306.962,A -85,B 0,C 180,E1 -29567.119,E2 -29567.119} C_VEL
LIN {X 0,Y 47.732,Z 307.59,A -85,B 0,C 180,E1 -29573.914,E2 -29573.914} C_VEL
LIN {X 0,Y 44.721,Z 307.825,A -85,B 0,C 180,E1 -29581.868,E2 -29581.868} C_VEL
LIN {X 0,Y 41.599,Z 307.081,A -85,B 0,C 180,E1 -29600.27,E2 -29600.27} C_VEL
LIN {X 0,Y 41.54,Z 306.126,A -85,B 0,C 180,E1 -29609.997,E2 -29609.997} C_VEL
LIN {X 0,Y 41.555,Z 304.703,A -85,B 0,C 180,E1 -29619.734,E2 -29619.734} C_VEL
LIN {X 0,Y 43.434,Z 301.712,A -85,B 0,C 180,E1 -29633.858,E2 -29633.858} C_VEL
LIN {X 0,Y 47.529,Z 297.657,A -85,B 0,C 180,E1 -29646.259,E2 -29646.259} C_VEL
LIN {X 0,Y 54.602,Z 291.418,A -85,B 0,C 180,E1 -29657.737,E2 -29657.737} C_VEL
LIN {X 0,Y 59.408,Z 287.071,A -85,B 0,C 180,E1 -29662.987,E2 -29662.987} C_VEL
LIN {X 0,Y 67.331,Z 279.168,A -85,B 0,C 180,E1 -29669.441,E2 -29669.441} C_VEL
LIN {X 0,Y 74.486,Z 271.103,A -85,B 0,C 180,E1 -29673.68,E2 -29673.68} C_VEL
LIN {X 0,Y 82.075,Z 261.286,A -85,B 0,C 180,E1 -29676.998,E2 -29676.998} C_VEL
LIN {X 0,Y 89.034,Z 250.32,A -85,B 0,C 180,E1 -29679.61,E2 -29679.61} C_VEL
LIN {X 0,Y 94.62,Z 239.593,A -85,B 0,C 180,E1 -29681.262,E2 -29681.262} C_VEL
LIN {X 0,Y 99.468,Z 227.799,A -85,B 0,C 180,E1 -29682.523,E2 -29682.523} C_VEL
LIN {X 0,Y 103.374,Z 214.651,A -85,B 0,C 180,E1 -29683.602,E2 -29683.602} C_VEL
LIN {X 0,Y 105.791,Z 202.259,A -85,B 0,C 180,E1 -29684.221,E2 -29684.221} C_VEL
LIN {X 0,Y 107.819,Z 184.232,A -85,B 0,C 180,E1 -29684.887,E2 -29684.887} C_VEL
LIN {X 0,Y 106.117,Z 179.287,A -85,B 0,C 180,E1 -29689.024,E2 -29689.024} C_VEL
LIN {X 0,Y 104.626,Z 175.349,A -85,B 0,C 180,E1 -29693.976,E2 -29693.976} C_VEL
LIN {X 0,Y 103.808,Z 172.458,A -85,B 0,C 180,E1 -29699.031,E2 -29699.031} C_VEL
LIN {X 0,Y 103.524,Z 172.344,A -85,B 0,C 180,E1 -29705.846,E2 -29705.846} C_VEL
LIN {X 0,Y 103.805,Z 172.849,A -85,B 0,C 180,E1 -29708.947,E2 -29708.947} C_VEL
LIN {X 0,Y 105.031,Z 176.56,A -85,B 0,C 180,E1 -29715.341,E2 -29715.341} C_VEL
LIN {X 0,Y 106.535,Z 180.536,A -85,B 0,C 180,E1 -29719.812,E2 -29719.812} C_VEL
LIN {X 0,Y 107.765,Z 184.225,A -85,B 0,C 180,E1 -29722.728,E2 -29722.728} C_VEL
LIN {X 0,Y 105.436,Z 203.153,A -85,B 0,C 180,E1 -29723.517,E2 -29723.517} C_VEL
LIN {X 0,Y 102.562,Z 216.092,A -85,B 0,C 180,E1 -29724.397,E2 -29724.397} C_VEL
LIN {X 0,Y 98.497,Z 228.593,A -85,B 0,C 180,E1 -29725.737,E2 -29725.737} C_VEL
LIN {X 0,Y 98.004,Z 229.869,A -85,B 0,C 180,E1 -29725.904,E2 -29725.904} C_VEL
LIN {X 0,Y 95.568,Z 235.218,A -85,B 0,C 180,E1 -29726.283,E2 -29726.283} C_VEL
LIN {X 0,Y 90.446,Z 243.706,A -85,B 0,C 180,E1 -29726.003,E2 -29726.003} C_VEL
LIN {X 0,Y 84.69,Z 251.792,A -85,B 0,C 180,E1 -29725.834,E2 -29725.834} C_VEL
LIN {X 0,Y 81.261,Z 256.509,A -85,B 0,C 180,E1 -29726.514,E2 -29726.514} C_VEL
LIN {X 0,Y 74.444,Z 265.437,A -85,B 0,C 180,E1 -29729.163,E2 -29729.163} C_VEL
LIN {X 0,Y 65.476,Z 275.282,A -85,B 0,C 180,E1 -29733.712,E2 -29733.712} C_VEL
LIN {X 0,Y 56.967,Z 283.209,A -85,B 0,C 180,E1 -29739.554,E2 -29739.554} C_VEL
LIN {X 0,Y 50.442,Z 288.569,A -85,B 0,C 180,E1 -29745.845,E2 -29745.845} C_VEL
LIN {X 0,Y 43.624,Z 293.819,A -85,B 0,C 180,E1 -29755.68,E2 -29755.68} C_VEL
LIN {X 0,Y 38.361,Z 297.913,A -85,B 0,C 180,E1 -29768.508,E2 -29768.508} C_VEL
LIN {X 0,Y 35.459,Z 300.66,A -85,B 0,C 180,E1 -29782.331,E2 -29782.331} C_VEL
LIN {X 0,Y 34.51,Z 303.09,A -85,B 0,C 180,E1 -29801.754,E2 -29801.754} C_VEL
LIN {X 0,Y 35.647,Z 304.015,A -85,B 0,C 180,E1 -29813.227,E2 -29813.227} C_VEL
LIN {X 0,Y 37.984,Z 304.518,A -85,B 0,C 180,E1 -29823.72,E2 -29823.72} C_VEL
LIN {X 0,Y 45.71,Z 304.311,A -85,B 0,C 180,E1 -29840.248,E2 -29840.248} C_VEL
LIN {X 0,Y 50.594,Z 303.629,A -85,B 0,C 180,E1 -29846.46,E2 -29846.46} C_VEL
LIN {X 0,Y 55.892,Z 302.514,A -85,B 0,C 180,E1 -29851.672,E2 -29851.672} C_VEL
LIN {X 0,Y 61.567,Z 300.97,A -85,B 0,C 180,E1 -29855.959,E2 -29855.959} C_VEL
LIN {X 0,Y 70.594,Z 297.838,A -85,B 0,C 180,E1 -29861.051,E2 -29861.051} C_VEL
LIN {X 0,Y 80.043,Z 293.621,A -85,B 0,C 180,E1 -29864.985,E2 -29864.985} C_VEL
LIN {X 0,Y 91.434,Z 287.186,A -85,B 0,C 180,E1 -29868.532,E2 -29868.532} C_VEL
LIN {X 0,Y 101.412,Z 280.085,A -85,B 0,C 180,E1 -29870.957,E2 -29870.957} C_VEL
LIN {X 0,Y 111.691,Z 271.017,A -85,B 0,C 180,E1 -29873.088,E2 -29873.088} C_VEL
LIN {X 0,Y 120.023,Z 262.03,A -85,B 0,C 180,E1 -29874.537,E2 -29874.537} C_VEL
LIN {X 0,Y 127.763,Z 251.825,A -85,B 0,C 180,E1 -29875.591,E2 -29875.591} C_VEL
LIN {X 0,Y 134.95,Z 239.924,A -85,B 0,C 180,E1 -29876.512,E2 -29876.512} C_VEL
LIN {X 0,Y 140.721,Z 227.516,A -85,B 0,C 180,E1 -29877.282,E2 -29877.282} C_VEL
LIN {X 0,Y 141.91,Z 224.39,A -85,B 0,C 180,E1 -29877.421,E2 -29877.421} C_VEL
LIN {X 0,Y 142.369,Z 222.992,A -85,B 0,C 180,E1 -29877.806,E2 -29877.806} C_VEL
LIN {X 0,Y 142.503,Z 221.562,A -85,B 0,C 180,E1 -29879.999,E2 -29879.999} C_VEL
LIN {X 0,Y 142.46,Z 221.224,A -85,B 0,C 180,E1 -29882.827,E2 -29882.827} C_VEL
LIN {X 0,Y 142.555,Z 221.539,A -85,B 0,C 180,E1 -29885.658,E2 -29885.658} C_VEL
LIN {X 0,Y 142.618,Z 222.991,A -85,B 0,C 180,E1 -29888.501,E2 -29888.501} C_VEL
LIN {X 0,Y 142.242,Z 224.297,A -85,B 0,C 180,E1 -29888.813,E2 -29888.813} C_VEL
LIN {X 0,Y 137.051,Z 236.628,A -85,B 0,C 180,E1 -29889.293,E2 -29889.293} C_VEL
LIN {X 0,Y 131.073,Z 247.607,A -85,B 0,C 180,E1 -29889.847,E2 -29889.847} C_VEL
LIN {X 0,Y 124.213,Z 257.757,A -85,B 0,C 180,E1 -29890.549,E2 -29890.549} C_VEL
LIN {X 0,Y 116.549,Z 267.093,A -85,B 0,C 180,E1 -29891.506,E2 -29891.506} C_VEL
LIN {X 0,Y 108.085,Z 275.622,A -85,B 0,C 180,E1 -29892.745,E2 -29892.745} C_VEL
LIN {X 0,Y 98.036,Z 283.936,A -85,B 0,C 180,E1 -29894.577,E2 -29894.577} C_VEL
LIN {X 0,Y 88.114,Z 290.657,A -85,B 0,C 180,E1 -29896.833,E2 -29896.833} C_VEL
LIN {X 0,Y 78.423,Z 296.047,A -85,B 0,C 180,E1 -29899.779,E2 -29899.779} C_VEL
LIN {X 0,Y 69.048,Z 300.277,A -85,B 0,C 180,E1 -29903.64,E2 -29903.64} C_VEL
LIN {X 0,Y 63.003,Z 302.536,A -85,B 0,C 180,E1 -29906.819,E2 -29906.819} C_VEL
LIN {X 0,Y 57.21,Z 304.325,A -85,B 0,C 180,E1 -29910.689,E2 -29910.689} C_VEL
LIN {X 0,Y 46.667,Z 306.689,A -85,B 0,C 180,E1 -29921.146,E2 -29921.146} C_VEL
LIN {X 0,Y 42.177,Z 307.297,A -85,B 0,C 180,E1 -29928.196,E2 -29928.196} C_VEL
LIN {X 0,Y 38.58,Z 307.493,A -85,B 0,C 180,E1 -29936.869,E2 -29936.869} C_VEL
LIN {X 0,Y 34.605,Z 306.71,A -85,B 0,C 180,E1 -29958.279,E2 -29958.279} C_VEL
LIN {X 0,Y 34.427,Z 305.736,A -85,B 0,C 180,E1 -29969.996,E2 -29969.996} C_VEL
LIN {X 0,Y 34.546,Z 304.273,A -85,B 0,C 180,E1 -29981.735,E2 -29981.735} C_VEL
LIN {X 0,Y 37.025,Z 301.245,A -85,B 0,C 180,E1 -29998.326,E2 -29998.326} C_VEL
LIN {X 0,Y 41.987,Z 297.145,A -85,B 0,C 180,E1 -30012.028,E2 -30012.028} C_VEL
LIN {X 0,Y 50.084,Z 290.849,A -85,B 0,C 180,E1 -30023.787,E2 -30023.787} C_VEL
LIN {X 0,Y 54.035,Z 287.63,A -85,B 0,C 180,E1 -30027.647,E2 -30027.647} C_VEL
LIN {X 0,Y 59.309,Z 282.965,A -85,B 0,C 180,E1 -30031.979,E2 -30031.979} C_VEL
LIN {X 0,Y 68.519,Z 273.781,A -85,B 0,C 180,E1 -30037.385,E2 -30037.385} C_VEL
LIN {X 0,Y 76.327,Z 264.654,A -85,B 0,C 180,E1 -30040.695,E2 -30040.695} C_VEL
LIN {X 0,Y 83.566,Z 254.589,A -85,B 0,C 180,E1 -30043.064,E2 -30043.064} C_VEL
LIN {X 0,Y 90.118,Z 243.389,A -85,B 0,C 180,E1 -30044.809,E2 -30044.809} C_VEL
LIN {X 0,Y 95.778,Z 231.148,A -85,B 0,C 180,E1 -30046.1,E2 -30046.1} C_VEL
LIN {X 0,Y 100.075,Z 218.423,A -85,B 0,C 180,E1 -30047.148,E2 -30047.148} C_VEL
LIN {X 0,Y 103.115,Z 205.174,A -85,B 0,C 180,E1 -30047.815,E2 -30047.815} C_VEL
LIN {X 0,Y 105.337,Z 188.146,A -85,B 0,C 180,E1 -30048.321,E2 -30048.321} C_VEL
LIN {X 0,Y 104.257,Z 184.502,A -85,B 0,C 180,E1 -30051.765,E2 -30051.765} C_VEL
LIN {X 0,Y 103.352,Z 181.791,A -85,B 0,C 180,E1 -30055.613,E2 -30055.613} C_VEL
LIN {X 0,Y 102.823,Z 179.368,A -85,B 0,C 180,E1 -30060.001,E2 -30060.001} C_VEL
LIN {X 0,Y 102.723,Z 179.495,A -85,B 0,C 180,E1 -30066.877,E2 -30066.877} C_VEL
LIN {X 0,Y 102.857,Z 180.01,A -85,B 0,C 180,E1 -30068.535,E2 -30068.535} C_VEL
LIN {X 0,Y 103.797,Z 183.278,A -85,B 0,C 180,E1 -30074.224,E2 -30074.224} C_VEL
LIN {X 0,Y 104.942,Z 186.864,A -85,B 0,C 180,E1 -30078.235,E2 -30078.235} C_VEL
LIN {X 0,Y 105.288,Z 188.065,A -85,B 0,C 180,E1 -30079.263,E2 -30079.263} C_VEL
LIN {X 0,Y 103.04,Z 204.535,A -85,B 0,C 180,E1 -30079.851,E2 -30079.851} C_VEL
LIN {X 0,Y 100.261,Z 216.411,A -85,B 0,C 180,E1 -30080.605,E2 -30080.605} C_VEL
LIN {X 0,Y 96.444,Z 227.934,A -85,B 0,C 180,E1 -30081.706,E2 -30081.706} C_VEL
LIN {X 0,Y 90.906,Z 240.4,A -85,B 0,C 180,E1 -30083.359,E2 -30083.359} C_VEL
LIN {X 0,Y 84.563,Z 251.539,A -85,B 0,C 180,E1 -30085.339,E2 -30085.339} C_VEL
LIN {X 0,Y 81.261,Z 256.509,A -85,B 0,C 180,E1 -30086.514,E2 -30086.514} C_VEL
LIN {X 0,Y 77.684,Z 261.074,A -85,B 0,C 180,E1 -30087.307,E2 -30087.307} C_VEL
LIN {X 0,Y 70.742,Z 268.177,A -85,B 0,C 180,E1 -30087.612,E2 -30087.612} C_VEL
LIN {X 0,Y 63.363,Z 274.768,A -85,B 0,C 180,E1 -30088.179,E2 -30088.179} C_VEL
LIN {X 0,Y 59.07,Z 278.486,A -85,B 0,C 180,E1 -30089.676,E2 -30089.676} C_VEL
LIN {X 0,Y 49.845,Z 286.056,A -85,B 0,C 180,E1 -30095.837,E2 -30095.837} C_VEL
LIN {X 0,Y 40.399,Z 292.735,A -85,B 0,C 180,E1 -30105.908,E2 -30105.908} C_VEL
LIN {X 0,Y 33.703,Z 297.147,A -85,B 0,C 180,E1 -30118.583,E2 -30118.583} C_VEL
LIN {X 0,Y 28.722,Z 300.8,A -85,B 0,C 180,E1 -30138.187,E2 -30138.187} C_VEL
LIN {X 0,Y 27.563,Z 302.19,A -85,B 0,C 180,E1 -30150.004,E2 -30150.004} C_VEL
LIN {X 0,Y 27.534,Z 303.485,A -85,B 0,C 180,E1 -30164.793,E2 -30164.793} C_VEL
LIN {X 0,Y 29.192,Z 304.386,A -85,B 0,C 180,E1 -30178.789,E2 -30178.789} C_VEL
LIN {X 0,Y 36.489,Z 304.921,A -85,B 0,C 180,E1 -30200.397,E2 -30200.397} C_VEL
LIN {X 0,Y 46.995,Z 303.899,A -85,B 0,C 180,E1 -30213.811,E2 -30213.811} C_VEL
LIN {X 0,Y 52.848,Z 302.747,A -85,B 0,C 180,E1 -30218.581,E2 -30218.581} C_VEL
LIN {X 0,Y 59.002,Z 301.181,A -85,B 0,C 180,E1 -30222.355,E2 -30222.355} C_VEL
LIN {X 0,Y 68.591,Z 298.005,A -85,B 0,C 180,E1 -30226.762,E2 -30226.762} C_VEL
LIN {X 0,Y 78.487,Z 293.74,A -85,B 0,C 180,E1 -30230.065,E2 -30230.065} C_VEL
LIN {X 0,Y 88.581,Z 288.262,A -85,B 0,C 180,E1 -30232.645,E2 -30232.645} C_VEL
LIN {X 0,Y 98.816,Z 281.388,A -85,B 0,C 180,E1 -30234.706,E2 -30234.706} C_VEL
LIN {X 0,Y 107.715,Z 274.072,A -85,B 0,C 180,E1 -30236.258,E2 -30236.258} C_VEL
LIN {X 0,Y 116.075,Z 265.784,A -85,B 0,C 180,E1 -30237.494,E2 -30237.494} C_VEL
LIN {X 0,Y 123.045,Z 257.535,A -85,B 0,C 180,E1 -30238.328,E2 -30238.328} C_VEL
LIN {X 0,Y 130.037,Z 247.507,A -85,B 0,C 180,E1 -30239.072,E2 -30239.072} C_VEL
LIN {X 0,Y 136.802,Z 235.272,A -85,B 0,C 180,E1 -30239.797,E2 -30239.797} C_VEL
LIN {X 0,Y 139.211,Z 229.978,A -85,B 0,C 180,E1 -30240.067,E2 -30240.067} C_VEL
LIN {X 0,Y 139.966,Z 228.178,A -85,B 0,C 180,E1 -30240.359,E2 -30240.359} C_VEL
LIN {X 0,Y 139.984,Z 227.877,A -85,B 0,C 180,E1 -30242.877,E2 -30242.877} C_VEL
LIN {X 0,Y 140.028,Z 228.35,A -85,B 0,C 180,E1 -30245.76,E2 -30245.76} C_VEL
LIN {X 0,Y 139.844,Z 228.934,A -85,B 0,C 180,E1 -30246.088,E2 -30246.088} C_VEL
LIN {X 0,Y 134.387,Z 240.485,A -85,B 0,C 180,E1 -30246.457,E2 -30246.457} C_VEL
LIN {X 0,Y 127.445,Z 251.968,A -85,B 0,C 180,E1 -30246.957,E2 -30246.957} C_VEL
LIN {X 0,Y 119.647,Z 262.327,A -85,B 0,C 180,E1 -30247.588,E2 -30247.588} C_VEL
LIN {X 0,Y 111.903,Z 270.803,A -85,B 0,C 180,E1 -30248.432,E2 -30248.432} C_VEL
LIN {X 0,Y 101.613,Z 280.009,A -85,B 0,C 180,E1 -30249.729,E2 -30249.729} C_VEL
LIN {X 0,Y 91.397,Z 287.429,A -85,B 0,C 180,E1 -30251.352,E2 -30251.352} C_VEL
LIN {X 0,Y 79.626,Z 294.295,A -85,B 0,C 180,E1 -30253.853,E2 -30253.853} C_VEL
LIN {X 0,Y 69.743,Z 298.849,A -85,B 0,C 180,E1 -30256.795,E2 -30256.795} C_VEL
LIN {X 0,Y 60.118,Z 302.336,A -85,B 0,C 180,E1 -30260.73,E2 -30260.73} C_VEL
LIN {X 0,Y 53.928,Z 304.093,A -85,B 0,C 180,E1 -30264.175,E2 -30264.175} C_VEL
LIN {X 0,Y 42.317,Z 306.416,A -85,B 0,C 180,E1 -30273.855,E2 -30273.855} C_VEL
LIN {X 0,Y 37.164,Z 306.997,A -85,B 0,C 180,E1 -30280.845,E2 -30280.845} C_VEL
LIN {X 0,Y 29.569,Z 306.941,A -85,B 0,C 180,E1 -30301.612,E2 -30301.612} C_VEL
LIN {X 0,Y 27.669,Z 306.339,A -85,B 0,C 180,E1 -30315.281,E2 -30315.281} C_VEL
LIN {X 0,Y 27.333,Z 305.347,A -85,B 0,C 180,E1 -30329.996,E2 -30329.996} C_VEL
LIN {X 0,Y 27.616,Z 303.842,A -85,B 0,C 180,E1 -30344.739,E2 -30344.739} C_VEL
LIN {X 0,Y 30.919,Z 300.77,A -85,B 0,C 180,E1 -30364.625,E2 -30364.625} C_VEL
LIN {X 0,Y 37,Z 296.625,A -85,B 0,C 180,E1 -30379.44,E2 -30379.44} C_VEL
LIN {X 0,Y 46.234,Z 290.28,A -85,B 0,C 180,E1 -30390.928,E2 -30390.928} C_VEL
LIN {X 0,Y 53.668,Z 284.483,A -85,B 0,C 180,E1 -30396.869,E2 -30396.869} C_VEL
LIN {X 0,Y 62.894,Z 276.287,A -85,B 0,C 180,E1 -30401.766,E2 -30401.766} C_VEL
LIN {X 0,Y 70.985,Z 267.778,A -85,B 0,C 180,E1 -30404.859,E2 -30404.859} C_VEL
LIN {X 0,Y 79.271,Z 257.266,A -85,B 0,C 180,E1 -30407.216,E2 -30407.216} C_VEL
LIN {X 0,Y 85.975,Z 246.852,A -85,B 0,C 180,E1 -30408.787,E2 -30408.787} C_VEL
LIN {X 0,Y 91.908,Z 235.445,A -85,B 0,C 180,E1 -30409.901,E2 -30409.901} C_VEL
LIN {X 0,Y 96.72,Z 223.198,A -85,B 0,C 180,E1 -30410.806,E2 -30410.806} C_VEL
LIN {X 0,Y 99.988,Z 211.799,A -85,B 0,C 180,E1 -30411.386,E2 -30411.386} C_VEL
LIN {X 0,Y 102.398,Z 198.738,A -85,B 0,C 180,E1 -30411.837,E2 -30411.837} C_VEL
LIN {X 0,Y 103.199,Z 192.078,A -85,B 0,C 180,E1 -30412.038,E2 -30412.038} C_VEL
LIN {X 0,Y 102.276,Z 188.607,A -85,B 0,C 180,E1 -30416.554,E2 -30416.554} C_VEL
LIN {X 0,Y 101.904,Z 186.371,A -85,B 0,C 180,E1 -30420.495,E2 -30420.495} C_VEL
LIN {X 0,Y 101.874,Z 186.619,A -85,B 0,C 180,E1 -30427.184,E2 -30427.184} C_VEL
LIN {X 0,Y 102.637,Z 190.099,A -85,B 0,C 180,E1 -30433.238,E2 -30433.238} C_VEL
LIN {X 0,Y 103.155,Z 192.103,A -85,B 0,C 180,E1 -30435.552,E2 -30435.552} C_VEL
LIN {X 0,Y 101.099,Z 205.885,A -85,B 0,C 180,E1 -30436.056,E2 -30436.056} C_VEL
LIN {X 0,Y 98.031,Z 218.011,A -85,B 0,C 180,E1 -30436.753,E2 -30436.753} C_VEL
LIN {X 0,Y 94.07,Z 229.246,A -85,B 0,C 180,E1 -30437.723,E2 -30437.723} C_VEL
LIN {X 0,Y 88.34,Z 241.515,A -85,B 0,C 180,E1 -30439.143,E2 -30439.143} C_VEL
LIN {X 0,Y 81.795,Z 252.49,A -85,B 0,C 180,E1 -30440.872,E2 -30440.872} C_VEL
LIN {X 0,Y 74.495,Z 262.376,A -85,B 0,C 180,E1 -30443.102,E2 -30443.102} C_VEL
LIN {X 0,Y 66.507,Z 271.358,A -85,B 0,C 180,E1 -30446.079,E2 -30446.079} C_VEL
LIN {X 0,Y 59.07,Z 278.486,A -85,B 0,C 180,E1 -30449.676,E2 -30449.676} C_VEL
LIN {X 0,Y 54.663,Z 282.039,A -85,B 0,C 180,E1 -30451.495,E2 -30451.495} C_VEL
LIN {X 0,Y 46.454,Z 287.365,A -85,B 0,C 180,E1 -30453.467,E2 -30453.467} C_VEL
LIN {X 0,Y 38.016,Z 292.048,A -85,B 0,C 180,E1 -30456.566,E2 -30456.566} C_VEL
LIN {X 0,Y 33.441,Z 294.552,A -85,B 0,C 180,E1 -30460.932,E2 -30460.932} C_VEL
LIN {X 0,Y 25.672,Z 298.865,A -85,B 0,C 180,E1 -30476.808,E2 -30476.808} C_VEL
LIN {X 0,Y 22.225,Z 300.941,A -85,B 0,C 180,E1 -30491.572,E2 -30491.572} C_VEL
LIN {X 0,Y 20.426,Z 302.604,A -85,B 0,C 180,E1 -30510.006,E2 -30510.006} C_VEL
LIN {X 0,Y 20.681,Z 303.88,A -85,B 0,C 180,E1 -30529.872,E2 -30529.872} C_VEL
LIN {X 0,Y 23.151,Z 304.749,A -85,B 0,C 180,E1 -30547.389,E2 -30547.389} C_VEL
LIN {X 0,Y 32.392,Z 305.235,A -85,B 0,C 180,E1 -30570.22,E2 -30570.22} C_VEL
LIN {X 0,Y 41.869,Z 304.477,A -85,B 0,C 180,E1 -30580.382,E2 -30580.382} C_VEL
LIN {X 0,Y 50.665,Z 302.98,A -85,B 0,C 180,E1 -30586.177,E2 -30586.177} C_VEL
LIN {X 0,Y 60.564,Z 300.439,A -85,B 0,C 180,E1 -30590.54,E2 -30590.54} C_VEL
LIN {X 0,Y 70.709,Z 296.869,A -85,B 0,C 180,E1 -30593.705,E2 -30593.705} C_VEL
LIN {X 0,Y 81.021,Z 292.16,A -85,B 0,C 180,E1 -30596.01,E2 -30596.01} C_VEL
LIN {X 0,Y 93.173,Z 285.054,A -85,B 0,C 180,E1 -30598.118,E2 -30598.118} C_VEL
LIN {X 0,Y 103.668,Z 277.266,A -85,B 0,C 180,E1 -30599.61,E2 -30599.61} C_VEL
LIN {X 0,Y 112.458,Z 269.268,A -85,B 0,C 180,E1 -30600.684,E2 -30600.684} C_VEL
LIN {X 0,Y 120.397,Z 260.552,A -85,B 0,C 180,E1 -30601.481,E2 -30601.481} C_VEL
LIN {X 0,Y 128.349,Z 249.856,A -85,B 0,C 180,E1 -30602.099,E2 -30602.099} C_VEL
LIN {X 0,Y 134.625,Z 239.345,A -85,B 0,C 180,E1 -30602.599,E2 -30602.599} C_VEL
LIN {X 0,Y 137.122,Z 234.388,A -85,B 0,C 180,E1 -30602.937,E2 -30602.937} C_VEL
LIN {X 0,Y 136.818,Z 235.029,A -85,B 0,C 180,E1 -30603.311,E2 -30603.311} C_VEL
LIN {X 0,Y 130.276,Z 246.938,A -85,B 0,C 180,E1 -30603.592,E2 -30603.592} C_VEL
LIN {X 0,Y 123.29,Z 257.088,A -85,B 0,C 180,E1 -30603.982,E2 -30603.982} C_VEL
LIN {X 0,Y 116.306,Z 265.456,A -85,B 0,C 180,E1 -30604.392,E2 -30604.392} C_VEL
LIN {X 0,Y 107.605,Z 274.17,A -85,B 0,C 180,E1 -30605.097,E2 -30605.097} C_VEL
LIN {X 0,Y 97.184,Z 282.661,A -85,B 0,C 180,E1 -30606.078,E2 -30606.078} C_VEL
LIN {X 0,Y 86.813,Z 289.495,A -85,B 0,C 180,E1 -30607.371,E2 -30607.371} C_VEL
LIN {X 0,Y 74.814,Z 295.799,A -85,B 0,C 180,E1 -30609.463,E2 -30609.463} C_VEL
LIN {X 0,Y 64.662,Z 299.938,A -85,B 0,C 180,E1 -30611.978,E2 -30611.978} C_VEL
LIN {X 0,Y 57.978,Z 302.127,A -85,B 0,C 180,E1 -30614.119,E2 -30614.119} C_VEL
LIN {X 0,Y 44.985,Z 305.193,A -85,B 0,C 180,E1 -30620.378,E2 -30620.378} C_VEL
LIN {X 0,Y 38.801,Z 306.144,A -85,B 0,C 180,E1 -30625.081,E2 -30625.081} C_VEL
LIN {X 0,Y 32.944,Z 306.691,A -85,B 0,C 180,E1 -30631.419,E2 -30631.419} C_VEL
LIN {X 0,Y 23.546,Z 306.59,A -85,B 0,C 180,E1 -30653.342,E2 -30653.342} C_VEL
LIN {X 0,Y 20.872,Z 305.97,A -85,B 0,C 180,E1 -30670.317,E2 -30670.317} C_VEL
LIN {X 0,Y 20.223,Z 304.949,A -85,B 0,C 180,E1 -30689.994,E2 -30689.994} C_VEL
LIN {X 0,Y 20.797,Z 303.41,A -85,B 0,C 180,E1 -30709.745,E2 -30709.745} C_VEL
LIN {X 0,Y 25.353,Z 300.293,A -85,B 0,C 180,E1 -30733.862,E2 -30733.862} C_VEL
LIN {X 0,Y 32.817,Z 296.106,A -85,B 0,C 180,E1 -30748.933,E2 -30748.933} C_VEL
LIN {X 0,Y 43.225,Z 289.712,A -85,B 0,C 180,E1 -30759.204,E2 -30759.204} C_VEL
LIN {X 0,Y 51.139,Z 283.972,A -85,B 0,C 180,E1 -30764.146,E2 -30764.146} C_VEL
LIN {X 0,Y 61.035,Z 275.597,A -85,B 0,C 180,E1 -30768.157,E2 -30768.157} C_VEL
LIN {X 0,Y 69.462,Z 266.988,A -85,B 0,C 180,E1 -30770.557,E2 -30770.557} C_VEL
LIN {X 0,Y 77.148,Z 257.551,A -85,B 0,C 180,E1 -30772.162,E2 -30772.162} C_VEL
LIN {X 0,Y 84.017,Z 247.266,A -85,B 0,C 180,E1 -30773.373,E2 -30773.373} C_VEL
LIN {X 0,Y 90.065,Z 236.033,A -85,B 0,C 180,E1 -30774.208,E2 -30774.208} C_VEL
LIN {X 0,Y 94.58,Z 225.251,A -85,B 0,C 180,E1 -30774.83,E2 -30774.83} C_VEL
LIN {X 0,Y 98.375,Z 213.044,A -85,B 0,C 180,E1 -30775.366,E2 -30775.366} C_VEL
LIN {X 0,Y 100.955,Z 200.18,A -85,B 0,C 180,E1 -30775.734,E2 -30775.734} C_VEL
LIN {X 0,Y 101.441,Z 196.57,A -85,B 0,C 180,E1 -30775.904,E2 -30775.904} C_VEL
LIN {X 0,Y 101.07,Z 194.647,A -85,B 0,C 180,E1 -30779.005,E2 -30779.005} C_VEL
LIN {X 0,Y 100.976,Z 193.51,A -85,B 0,C 180,E1 -30780.998,E2 -30780.998} C_VEL
LIN {X 0,Y 100.924,Z 193.522,A -85,B 0,C 180,E1 -30785.997,E2 -30785.997} C_VEL
LIN {X 0,Y 101.396,Z 196.518,A -85,B 0,C 180,E1 -30791.675,E2 -30791.675} C_VEL
LIN {X 0,Y 100.181,Z 204.21,A -85,B 0,C 180,E1 -30792.003,E2 -30792.003} C_VEL
LIN {X 0,Y 96.978,Z 217.346,A -85,B 0,C 180,E1 -30792.604,E2 -30792.604} C_VEL
LIN {X 0,Y 93.01,Z 228.589,A -85,B 0,C 180,E1 -30793.384,E2 -30793.384} C_VEL
LIN {X 0,Y 87.127,Z 241.054,A -85,B 0,C 180,E1 -30794.548,E2 -30794.548} C_VEL
LIN {X 0,Y 80.386,Z 252.189,A -85,B 0,C 180,E1 -30795.911,E2 -30795.911} C_VEL
LIN {X 0,Y 73.689,Z 261.2,A -85,B 0,C 180,E1 -30797.5,E2 -30797.5} C_VEL
LIN {X 0,Y 65.36,Z 270.467,A -85,B 0,C 180,E1 -30799.809,E2 -30799.809} C_VEL
LIN {X 0,Y 55.565,Z 279.43,A -85,B 0,C 180,E1 -30803.515,E2 -30803.515} C_VEL
LIN {X 0,Y 46.063,Z 286.655,A -85,B 0,C 180,E1 -30808.686,E2 -30808.686} C_VEL
LIN {X 0,Y 38.521,Z 291.541,A -85,B 0,C 180,E1 -30814.82,E2 -30814.82} C_VEL
LIN {X 0,Y 33.441,Z 294.552,A -85,B 0,C 180,E1 -30820.932,E2 -30820.932} C_VEL
LIN {X 0,Y 29.013,Z 296.867,A -85,B 0,C 180,E1 -30826.723,E2 -30826.723} C_VEL
LIN {X 0,Y 24.214,Z 298.881,A -85,B 0,C 180,E1 -30832.946,E2 -30832.946} C_VEL
LIN {X 0,Y 15.327,Z 302.098,A -85,B 0,C 180,E1 -30855.098,E2 -30855.098} C_VEL
LIN {X 0,Y 13.229,Z 303.366,A -85,B 0,C 180,E1 -30877.223,E2 -30877.223} C_VEL
LIN {X 0,Y 13.275,Z 303.66,A -85,B 0,C 180,E1 -30885.703,E2 -30885.703} C_VEL
LIN {X 0,Y 17.986,Z 305.105,A -85,B 0,C 180,E1 -30921.41,E2 -30921.41} C_VEL
LIN {X 0,Y 29.49,Z 305.549,A -85,B 0,C 180,E1 -30942.428,E2 -30942.428} C_VEL
LIN {X 0,Y 39.083,Z 304.861,A -85,B 0,C 180,E1 -30949.638,E2 -30949.638} C_VEL
LIN {X 0,Y 49.441,Z 303.213,A -85,B 0,C 180,E1 -30954.321,E2 -30954.321} C_VEL
LIN {X 0,Y 59.804,Z 300.628,A -85,B 0,C 180,E1 -30957.352,E2 -30957.352} C_VEL
LIN {X 0,Y 70.284,Z 297.012,A -85,B 0,C 180,E1 -30959.544,E2 -30959.544} C_VEL
LIN {X 0,Y 80.839,Z 292.255,A -85,B 0,C 180,E1 -30961.108,E2 -30961.108} C_VEL
LIN {X 0,Y 89.082,Z 287.703,A -85,B 0,C 180,E1 -30962.092,E2 -30962.092} C_VEL
LIN {X 0,Y 87.707,Z 288.542,A -85,B 0,C 180,E1 -30962.578,E2 -30962.578} C_VEL
LIN {X 0,Y 77.461,Z 294.047,A -85,B 0,C 180,E1 -30963.578,E2 -30963.578} C_VEL
LIN {X 0,Y 67.028,Z 298.509,A -85,B 0,C 180,E1 -30965.044,E2 -30965.044} C_VEL
LIN {X 0,Y 56.664,Z 301.915,A -85,B 0,C 180,E1 -30967.123,E2 -30967.123} C_VEL
LIN {X 0,Y 43.025,Z 304.94,A -85,B 0,C 180,E1 -30971.442,E2 -30971.442} C_VEL
LIN {X 0,Y 36.358,Z 305.871,A -85,B 0,C 180,E1 -30974.861,E2 -30974.861} C_VEL
LIN {X 0,Y 29.856,Z 306.379,A -85,B 0,C 180,E1 -30979.666,E2 -30979.666} C_VEL
LIN {X 0,Y 18.327,Z 306.238,A -85,B 0,C 180,E1 -30999.907,E2 -30999.907} C_VEL
LIN {X 0,Y 14.365,Z 305.599,A -85,B 0,C 180,E1 -31020.7,E2 -31020.7} C_VEL
LIN {X 0,Y 13.112,Z 304.544,A -85,B 0,C 180,E1 -31049.991,E2 -31049.991} C_VEL
LIN {X 0,Y 14.279,Z 302.978,A -85,B 0,C 180,E1 -31079.475,E2 -31079.475} C_VEL
LIN {X 0,Y 20.796,Z 299.817,A -85,B 0,C 180,E1 -31107.648,E2 -31107.648} C_VEL
LIN {X 0,Y 29.771,Z 295.586,A -85,B 0,C 180,E1 -31120.769,E2 -31120.769} C_VEL
LIN {X 0,Y 41.235,Z 289.142,A -85,B 0,C 180,E1 -31128.515,E2 -31128.515} C_VEL
LIN {X 0,Y 48.135,Z 284.462,A -85,B 0,C 180,E1 -31131.606,E2 -31131.606} C_VEL
LIN {X 0,Y 58.251,Z 276.412,A -85,B 0,C 180,E1 -31134.461,E2 -31134.461} C_VEL
LIN {X 0,Y 66.914,Z 268.062,A -85,B 0,C 180,E1 -31136.16,E2 -31136.16} C_VEL
LIN {X 0,Y 75.63,Z 257.835,A -85,B 0,C 180,E1 -31137.354,E2 -31137.354} C_VEL
LIN {X 0,Y 82.62,Z 247.68,A -85,B 0,C 180,E1 -31138.147,E2 -31138.147} C_VEL
LIN {X 0,Y 88.75,Z 236.621,A -85,B 0,C 180,E1 -31138.669,E2 -31138.669} C_VEL
LIN {X 0,Y 93.691,Z 225.149,A -85,B 0,C 180,E1 -31139.118,E2 -31139.118} C_VEL
LIN {X 0,Y 97.542,Z 213.048,A -85,B 0,C 180,E1 -31139.486,E2 -31139.486} C_VEL
LIN {X 0,Y 99.983,Z 201.542,A -85,B 0,C 180,E1 -31139.862,E2 -31139.862} C_VEL
LIN {X 0,Y 99.956,Z 200.43,A -85,B 0,C 180,E1 -31142.016,E2 -31142.016} C_VEL
LIN {X 0,Y 99.927,Z 200.715,A -85,B 0,C 180,E1 -31145.981,E2 -31145.981} C_VEL
LIN {X 0,Y 99.928,Z 201.661,A -85,B 0,C 180,E1 -31147.797,E2 -31147.797} C_VEL
LIN {X 0,Y 96.915,Z 214.898,A -85,B 0,C 180,E1 -31148.314,E2 -31148.314} C_VEL
LIN {X 0,Y 92.494,Z 227.873,A -85,B 0,C 180,E1 -31148.974,E2 -31148.974} C_VEL
LIN {X 0,Y 87.35,Z 239.019,A -85,B 0,C 180,E1 -31149.74,E2 -31149.74} C_VEL
LIN {X 0,Y 80.461,Z 250.588,A -85,B 0,C 180,E1 -31150.695,E2 -31150.695} C_VEL
LIN {X 0,Y 72.736,Z 260.993,A -85,B 0,C 180,E1 -31151.962,E2 -31151.962} C_VEL
LIN {X 0,Y 65.019,Z 269.513,A -85,B 0,C 180,E1 -31153.397,E2 -31153.397} C_VEL
LIN {X 0,Y 56.524,Z 277.359,A -85,B 0,C 180,E1 -31155.511,E2 -31155.511} C_VEL
LIN {X 0,Y 46.433,Z 285.033,A -85,B 0,C 180,E1 -31158.926,E2 -31158.926} C_VEL
LIN {X 0,Y 34.971,Z 292.086,A -85,B 0,C 180,E1 -31165.272,E2 -31165.272} C_VEL
LIN {X 0,Y 25.709,Z 296.786,A -85,B 0,C 180,E1 -31174.913,E2 -31174.913} C_VEL
LIN {X 0,Y 16.228,Z 301.098,A -85,B 0,C 180,E1 -31200.026,E2 -31200.026} C_VEL
LIN {X 0,Y 13.275,Z 303.66,A -85,B 0,C 180,E1 -31245.703,E2 -31245.703} C_VEL
LIN {X 0,Y 14.578,Z 304.609,A -85,B 0,C 180,E1 -31269.286,E2 -31269.286} C_VEL
LIN {X 0,Y 19.409,Z 305.579,A -85,B 0,C 180,E1 -31298.923,E2 -31298.923} C_VEL
LIN {X 0,Y 25.412,Z 305.868,A -85,B 0,C 180,E1 -31312.448,E2 -31312.448} C_VEL
LIN {X 0,Y 30.794,Z 305.765,A -85,B 0,C 180,E1 -31317.539,E2 -31317.539} C_VEL
LIN {X 0,Y 32.707,Z 305.617,A -85,B 0,C 180,E1 -31318.423,E2 -31318.423} C_VEL
LIN {X 0,Y 42.18,Z 304.67,A -85,B 0,C 180,E1 -31321.268,E2 -31321.268} C_VEL
LIN {X 0,Y 42.194,Z 304.688,A -85,B 0,C 180,E1 -31321.937,E2 -31321.937} C_VEL
LIN {X 0,Y 35.211,Z 305.592,A -85,B 0,C 180,E1 -31323.592,E2 -31323.592} C_VEL
LIN {X 0,Y 21.421,Z 306.165,A -85,B 0,C 180,E1 -31330.147,E2 -31330.147} C_VEL
LIN {X 0,Y 8.874,Z 305.228,A -85,B 0,C 180,E1 -31357.608,E2 -31357.608} C_VEL
LIN {X 0,Y 5.984,Z 304.133,A -85,B 0,C 180,E1 -31409.98,E2 -31409.98} C_VEL
LIN {X 0,Y 11.612,Z 301.614,A -85,B 0,C 180,E1 -31475.185,E2 -31475.185} C_VEL
LIN {X 0,Y 21.37,Z 298.062,A -85,B 0,C 180,E1 -31490.578,E2 -31490.578} C_VEL
LIN {X 0,Y 31.699,Z 293.401,A -85,B 0,C 180,E1 -31496.052,E2 -31496.052} C_VEL
